# B&R Automation Studio project EFI (part 14)

#### FileManager.st
```iecst
ACTION FileManager:

	CASE Handling.Data.Step OF

		0:  (* link (create) a file device *)
			Handling.Functionblock.DevLink_0.enable := 1;
			Handling.Functionblock.DevLink_0.pDevice := ADR(Handling.Data.Device);  (* name of the device, which is needed for other functionblocks *)
			Handling.Functionblock.DevLink_0.pParam := ADR(Handling.Data.Parameter);  (* devicepath *)
			Handling.Functionblock.DevLink_0;  (* call the function*)

			IF Handling.Functionblock.DevLink_0.status = 0 THEN  (* DevLink successful *)
				Handling.Data.Step := 1;  (* next Step*)
				FolderHandling.Data.Step := 1;  (* next Step*)
			ELSIF Handling.Functionblock.DevLink_0.status = ERR_FUB_BUSY THEN  (* DevLink not finished -> redo *)
				(* Busy *)
			ELSIF Handling.Functionblock.DevLink_0.status = fiERR_SYSTEM THEN  (* DevLink error = fiERR_SYSTEM -> detailed info with function "FileIoGetSysError" *)
				(* get detail errorinformation *)
				Error := FileIoGetSysError();
				(* Goto Error Step *)
				Handling.Data.Step := 255;

				FolderError := FileIoGetSysError();
				FolderHandling.Data.Step := 255;
			ELSE  (* Goto Error Step *)
				Handling.Data.Step := 255;
				FolderHandling.Data.Step := 255;
			END_IF

		1:  (* Wait and comannd step *)
			IF Handling.Command.bCreateFile = 1 THEN
				(* Create a new file with the name from the variable "Handling.Data.FileName" *)
				Handling.Data.Step := 10;  (* next Step*)

			ELSIF Handling.Command.bWriteFile = 1 THEN
				(* writes the data from variable "Handling.Data.WriteData"
				   in the file with the name from the variable "Handling.Data.FileName" *)
				Handling.Data.Step := 20;  (* next Step*)

			ELSIF Handling.Command.bReadFile = 1 THEN
				(* read data to variable "Handling.Data.ReadData"
				   from the file with the name of the variable "Handling.Data.FileName" *)
				Handling.Data.Step := 30;  (* next Step*)

			ELSIF Handling.Command.bReadExFile = 1 THEN
				(* read data to variable "Handling.Data.ReadData"
				   from the file with the name of the variable "Handling.Data.FileName" *)
				Handling.Data.Step := 40;  (* next Step*)

			ELSIF Handling.Command.bCopyFile = 1 THEN
				(* creates a copy with the name from the variable "Handling.Data.NewFileName"
				   from the file with the name from the variable "Handling.Data.FileName" *)
				Handling.Data.Step := 50;  (* next Step*)

			ELSIF Handling.Command.bRenameFile = 1 THEN
				(* renames the the file with the name from the variable "Handling.Data.FileName"
				   to the name from the variable "Handling.Data.NewFileName" *)
				Handling.Data.Step := 60;  (* next Step*)

			ELSIF Handling.Command.bDeleteFile = 1 THEN
				(* deletes the file with the name from the variable "Handling.Data.FileName" *)
				Handling.Data.Step := 70;  (* next Step*)

			END_IF

			(***********************************************************************************************)
		10:  (* create a new File with the selected name  *)
			Handling.Functionblock.FileCreate_0.enable := 1;
			Handling.Functionblock.FileCreate_0.pDevice := ADR(Handling.Data.Device);  (* name of the linked device *)
			Handling.Functionblock.FileCreate_0.pFile := ADR(Handling.Data.FileName);  (* name of the file *)
			Handling.Functionblock.FileCreate_0;  (* call the function*)

			IF Handling.Functionblock.FileCreate_0.status = 0 THEN  (* FileCreate successful *)
				Handling.Data.Step := 11;  (* next Step*)
			ELSIF Handling.Functionblock.FileCreate_0.status = ERR_FUB_BUSY THEN  (* FileCreate not finished -> redo *)
				(* Busy *)
			ELSE  (* Goto Error Step *)
				Handling.Data.Step := 255;
			END_IF

		11:	 (* close file, because of limited number of available file handles on the system *)
			Handling.Functionblock.FileClose_0.enable := 1;
			Handling.Functionblock.FileClose_0.ident := Handling.Functionblock.FileCreate_0.ident; (* ident for FileCreate-functionblock*)
			Handling.Functionblock.FileClose_0;  (* call the function*)

			IF Handling.Functionblock.FileClose_0.status = 0 THEN  (* FileClose successful *)
				Handling.Data.Step := 1;  (* next Step*)
				Handling.Command.bCreateFile := 0;  (* clear command *)
			ELSIF Handling.Functionblock.FileClose_0.status = ERR_FUB_BUSY THEN  (* FileClose not finished -> redo *)
				(* Busy *)
			ELSE  (* Goto Error Step *)
				Handling.Data.Step := 255;
			END_IF

			(***********************************************************************************************)
		20:	(* open file for write access *)
			Handling.Functionblock.FileOpen_0.enable := 1;
			Handling.Functionblock.FileOpen_0.pDevice := ADR(Handling.Data.Device);  (* name of the linked device *)
			Handling.Functionblock.FileOpen_0.pFile :=  ADR(Handling.Data.FileName);  (* name of the file *)
			Handling.Functionblock.FileOpen_0.mode := fiWRITE_ONLY; (* write access *)
			Handling.Functionblock.FileOpen_0;  (* call the function*)

			IF Handling.Functionblock.FileOpen_0.status = 0 THEN  (* FileOpen successful *)
				Handling.Data.Step := 21;  (* next Step*)
			ELSIF Handling.Functionblock.FileOpen_0.status = ERR_FUB_BUSY THEN  (* FileOpen not finished -> redo *)
				(* Busy *)
			ELSE  (* Goto Error Step *)
				Handling.Data.Step := 255;
			END_IF

		21: (* write data into file *)
			Handling.Functionblock.FileWrite_0.enable := 1;
			Handling.Functionblock.FileWrite_0.ident := Handling.Functionblock.FileOpen_0.ident;
			Handling.Functionblock.FileWrite_0.offset := 0; (* start at the beginning of the file *)
			Handling.Functionblock.FileWrite_0.pSrc := ADR(Handling.Data.WriteData);
			Handling.Functionblock.FileWrite_0.len := strlen( ADR(Handling.Data.WriteData) );
			Handling.Functionblock.FileWrite_0;  (* call the function*)

			IF Handling.Functionblock.FileWrite_0.status = 0 THEN  (* FileWrite successful *)
				Handling.Data.Step := 22;  (* next Step*)
			ELSIF Handling.Functionblock.FileWrite_0.status = ERR_FUB_BUSY THEN  (* FileWrite not finished -> redo *)
				(* Busy *)
			ELSE  (* Goto Error Step *)
				Handling.Data.Step := 255;
			END_IF

		22:	 (* close file, because of limited number of available file handles on the system *)
			Handling.Functionblock.FileClose_0.enable := 1;
			Handling.Functionblock.FileClose_0.ident := Handling.Functionblock.FileOpen_0.ident; (* ident for FileCreate-functionblock*)
			Handling.Functionblock.FileClose_0;  (* call the function*)

			IF Handling.Functionblock.FileClose_0.status = 0 THEN  (* FileClose successful *)
				Handling.Data.Step := 1;  (* next Step*)
				Handling.Command.bWriteFile := 0;  (* clear command *)
			ELSIF Handling.Functionblock.FileClose_0.status = ERR_FUB_BUSY THEN  (* FileClose not finished -> redo *)
				(* Busy *)
			ELSE  (* Goto Error Step *)
				Handling.Data.Step := 255;
			END_IF

			(***********************************************************************************************)
		30:	(* open file for read access *)
			Handling.Functionblock.FileOpen_0.enable := 1;
			Handling.Functionblock.FileOpen_0.pDevice := ADR(Handling.Data.Device);  (* name of the linked device *)
			Handling.Functionblock.FileOpen_0.pFile :=  ADR(Handling.Data.FileName);  (* name of the file *)
			Handling.Functionblock.FileOpen_0.mode := fiREAD_ONLY;  (* read access *)
			Handling.Functionblock.FileOpen_0;  (* call the function*)

			IF Handling.Functionblock.FileOpen_0.status = 0 THEN  (* FileOpen successful *)
				Handling.Data.Step := 31;  (* next Step*)
			ELSIF Handling.Functionblock.FileOpen_0.status = ERR_FUB_BUSY THEN  (* FileOpen not finished -> redo *)
				(* Busy *)
			ELSE  (* Goto Error Step *)
				Handling.Data.Step := 255;
			END_IF

		31: (* read data from file *)
			Handling.Functionblock.FileRead_0.enable := 1;
			Handling.Functionblock.FileRead_0.ident := Handling.Functionblock.FileOpen_0.ident;  (* ident of the previous "FileOpen" *)
			Handling.Functionblock.FileRead_0.offset := 0;  (* start at the beginning of the file *)
			Handling.Functionblock.FileRead_0.pDest := ADR(Handling.Data.ReadData);  (* adress of the destination of reaaded datas *)
			Handling.Functionblock.FileRead_0.len := SIZEOF( Handling.Data.ReadData );  (* lenght of data, which should be readed *)
			Handling.Functionblock.FileRead_0;  (* call the function*)

			IF Handling.Functionblock.FileRead_0.status = 0 THEN  (* FileRead successful *)
				Handling.Data.Step := 32;  (* next Step*)
			ELSIF Handling.Functionblock.FileRead_0.status = ERR_FUB_BUSY THEN  (* FileRead not finished -> redo *)
				(* Busy *)
			ELSE  (* Goto Error Step *)
				Handling.Data.Step := 255;
			END_IF

		32:	 (* close file, because of limited number of available file handles on the system *)
			Handling.Functionblock.FileClose_0.enable := 1;
			Handling.Functionblock.FileClose_0.ident := Handling.Functionblock.FileOpen_0.ident; (* ident for FileCreate-functionblock*)
			Handling.Functionblock.FileClose_0;  (* call the function*)

			IF Handling.Functionblock.FileClose_0.status = 0 THEN  (* FileClose successful *)
				Handling.Data.Step := 1;  (* next Step*)
				Handling.Command.bReadFile := 0;  (* clear command *)
			ELSIF Handling.Functionblock.FileClose_0.status = ERR_FUB_BUSY THEN  (* FileClose not finished -> redo *)
				(* Busy *)
			ELSE  (* Goto Error Step *)
				Handling.Data.Step := 255;
			END_IF

			(***********************************************************************************************)
		40:	(* open file for read access *)
			Handling.Functionblock.FileOpen_0.enable := 1;
			Handling.Functionblock.FileOpen_0.pDevice := ADR(Handling.Data.Device);  (* name of the linked device *)
			Handling.Functionblock.FileOpen_0.pFile :=  ADR(Handling.Data.FileName);  (* name of the file *)
			Handling.Functionblock.FileOpen_0.mode := fiREAD_ONLY;  (* read access *)
			Handling.Functionblock.FileOpen_0;  (* call the function*)

			IF Handling.Functionblock.FileOpen_0.status = 0 THEN  (* FileOpen successful *)
				Handling.Data.Step := 41;  (* next Step*)
			ELSIF Handling.Functionblock.FileOpen_0.status = ERR_FUB_BUSY THEN  (* FileOpen not finished -> redo *)
				(* Busy *)
			ELSE  (* Goto Error Step *)
				Handling.Data.Step := 255;
			END_IF

		41: (* read data from file *)
			Handling.Functionblock.FileReadEx_0.enable := 1;
			Handling.Functionblock.FileReadEx_0.ident := Handling.Functionblock.FileOpen_0.ident;  (* ident of the previous "FileOpen" *)
			Handling.Functionblock.FileReadEx_0.offset := 0;  (* start at the beginning of the file *)
			Handling.Functionblock.FileReadEx_0.pDest := ADR(Handling.Data.ReadData);  (* adress of the destination of reaaded datas *)
			Handling.Functionblock.FileReadEx_0.len := SIZEOF( Handling.Data.ReadData );  (* lenght of data, which should be readed *)
			Handling.Functionblock.FileReadEx_0;  (* call the function*)

			IF Handling.Functionblock.FileReadEx_0.status = 0 THEN  (* FileReadEx successful *)
				(* Handling.Functionblock.FileReadEx_0.bytesread includes the lenght of the readed data *)
				Handling.Data.Step := 42;  (* next Step*)
			ELSIF Handling.Functionblock.FileReadEx_0.status = ERR_FUB_BUSY THEN  (* FileReadEx not finished -> redo *)
				(* Busy *)
			ELSE  (* Goto Error Step *)
				Handling.Data.Step := 255;
			END_IF

		42:	 (* close file, because of limited number of available file handles on the system *)
			Handling.Functionblock.FileClose_0.enable := 1;
			Handling.Functionblock.FileClose_0.ident := Handling.Functionblock.FileOpen_0.ident; (* ident for FileCreate-functionblock*)
			Handling.Functionblock.FileClose_0;  (* call the function*)

			IF Handling.Functionblock.FileClose_0.status = 0 THEN  (* FileClose successful *)
				Handling.Data.Step := 1;  (* next Step*)
				Handling.Command.bReadExFile := 0;  (* clear command *)
			ELSIF Handling.Functionblock.FileClose_0.status = ERR_FUB_BUSY THEN  (* FileClose not finished -> redo *)
				(* Busy *)
			ELSE  (* Goto Error Step *)
				Handling.Data.Step := 255;
			END_IF

			(***********************************************************************************************)
		50: (* copy a file *)

			Handling.Functionblock.FileCopy_0.enable := 1;
			Handling.Functionblock.FileCopy_0.option := fiOVERWRITE;  (* overwrite existing file *)
			Handling.Functionblock.FileCopy_0.pSrcDev := ADR(Handling.Data.Device);  (* name of a linked device *)
			Handling.Functionblock.FileCopy_0.pSrc := ADR(Handling.Data.FileName);  (* name of the source file *)
			Handling.Functionblock.FileCopy_0.pDestDev := ADR(Handling.Data.Device);  (* name of a linked device *)
			Handling.Functionblock.FileCopy_0.pDest := ADR(Handling.Data.NewFileName);  (* name of the new file*)
			Handling.Functionblock.FileCopy_0;  (* call the function*)

			IF Handling.Functionblock.FileCopy_0.status = 0 THEN  (* FileCopy successful *)
				Handling.Data.Step := 1;  (* next Step*)
				Handling.Command.bCopyFile := 0;  (* clear command *)
			ELSIF Handling.Functionblock.FileCopy_0.status = ERR_FUB_BUSY THEN  (* FileCopy not finished -> redo *)
				(* Busy *)
			ELSE  (* Goto Error Step *)
				Handling.Data.Step := 255;
			END_IF

			(***********************************************************************************************)
		60: (* rename a file *)

			Handling.Functionblock.FileRename_0.enable := 1;
			Handling.Functionblock.FileRename_0.pDevice := ADR(Handling.Data.Device);  (* name of the linked device *)
			Handling.Functionblock.FileRename_0.pName := ADR(Handling.Data.FileName);  (* actual file name *)
			Handling.Functionblock.FileRename_0.pNewName := ADR(Handling.Data.NewFileName);  (* new file name *)
			Handling.Functionblock.FileRename_0;  (* call the function*)

			IF Handling.Functionblock.FileRename_0.status = 0 THEN  (* FileRename successful *)
				Handling.Data.Step := 1;  (* next Step*)
				Handling.Command.bRenameFile := 0;  (* clear command *)
			ELSIF Handling.Functionblock.FileRename_0.status = ERR_FUB_BUSY THEN  (* FileRename not finished -> redo *)
				(* Busy *)
			ELSE  (* Goto Error Step *)
				Handling.Data.Step := 255;
			END_IF

			(***********************************************************************************************)
		70: (* delete a file *)

			Handling.Functionblock.FileDelete_0.enable := 1;
			Handling.Functionblock.FileDelete_0.pDevice := ADR(Handling.Data.Device);  (* name of a linked device *)
			Handling.Functionblock.FileDelete_0.pName := ADR(Handling.Data.FileName);  (* name of the source file *)
			Handling.Functionblock.FileDelete_0;  (* call the function*)

			IF Handling.Functionblock.FileDelete_0.status = 0 THEN  (* FileRename successful *)
				Handling.Data.Step := 1;  (* next Step*)
				Handling.Command.bDeleteFile := 0;  (* clear command *)
			ELSIF Handling.Functionblock.FileDelete_0.status = ERR_FUB_BUSY THEN  (* FileRename not finished -> redo *)
				(* Busy *)
			ELSE  (* Goto Error Step *)
				Handling.Data.Step := 255;
			END_IF

			(***********************************************************************************************)
		255:  (* Here some error Handling has to be implemented *)

	END_CASE

END_ACTION
```

#### FolderManager.st
```iecst
ACTION FolderManager:

	CASE FolderHandling.Data.Step OF

		0:  (* link (create) a file device *)
			//			FolderHandling.Functionblock.DevLink_0.enable := 1;
			//			FolderHandling.Functionblock.DevLink_0.pDevice := ADR(FolderHandling.Data.Device);  (* name of the device, which is needed for other functionblocks *)
			//			FolderHandling.Functionblock.DevLink_0.pParam := ADR(FolderHandling.Data.Parameter);  (* devicepath *)
			//			FolderHandling.Functionblock.DevLink_0;  (* call the function*)
			//
			//			IF FolderHandling.Functionblock.DevLink_0.status = 0 THEN  (* DevLink successful *)
			//				FolderHandling.Data.Step := 1;  (* next Step*)
			//			ELSIF FolderHandling.Functionblock.DevLink_0.status = ERR_FUB_BUSY THEN  (* DevLink not finished -> redo *)
			//				(* Busy *)
			//			ELSIF FolderHandling.Functionblock.DevLink_0.status = fiERR_SYSTEM THEN  (* DevLink FolderError = fiERR_SYSTEM -> detailed info with function "FileIoGetSysFolderError" *)
			//				(* get detail FolderErrorinformation *)
			//				FolderError := FileIoGetSysFolderError();
			//				(* Goto FolderError Step *)
			//				FolderHandling.Data.Step := 255;
			//			ELSE  (* Goto FolderError Step *)
			//				FolderHandling.Data.Step := 255;
			//			END_IF

		1:  (* Wait and comannd step *)
			IF FolderHandling.Command.bDirRead = 1 THEN
				(* read all names of files and folders into the string-array "FolderHandling.Data.FileList" *)
				FolderHandling.Data.Step := 10;  (* next Step*)

			ELSIF FolderHandling.Command.bDirCreate = 1 THEN
				(* creates a new directory with the name on the variable "FolderHandling.Data.DirName" *)
				FolderHandling.Data.Step := 20;  (* next Step*)

			ELSIF FolderHandling.Command.bDirCopy = 1 THEN
				(* copy a directory with the name on the variable "FolderHandling.Data.DirName"
				   to a directory with the name on the variable "FolderHandling.Data.NewDirName"*)
				FolderHandling.Data.Step := 30;  (* next Step*)

			ELSIF FolderHandling.Command.bDirRename = 1 THEN
				(* rename the directory with the name on the variable "FolderHandling.Data.DirName"
				   to the name on the variable "FolderHandling.Data.NewDirName"*)
				FolderHandling.Data.Step := 40;  (* next Step*)

			ELSIF FolderHandling.Command.bDirDelete = 1 THEN
				(* delete the directory with the name on the variable "FolderHandling.Data.DirName" *)
				FolderHandling.Data.Step := 50;  (* next Step*)

			ELSIF FolderHandling.Command.bDevMemInfo = 1 THEN
				(* read information about your device *)
				FolderHandling.Data.Step := 60;  (* next Step*)

			ELSIF FolderHandling.Command.bGetAttributes = 1 THEN
				(* read information about your device-settings *)
				FolderHandling.Data.Step := 70;  (* next Step*)

			ELSIF FolderHandling.Command.bSetAttributes = 1 THEN
				(* set device settings*)
				FolderHandling.Data.Step := 80;  (* next Step*)

			END_IF

			(***********************************************************************************************)
		10: (* calulate the number of files and directories *)
			FolderHandling.Functionblock.DirInfo_0.enable := 1;
			FolderHandling.Functionblock.DirInfo_0.pDevice := ADR(FolderHandling.Data.Device);  (* name of the device *)
			FolderHandling.Functionblock.DirInfo_0.pPath := 0;
			FolderHandling.Functionblock.DirInfo_0;  (* call the function*)

			IF FolderHandling.Functionblock.DirInfo_0.status = 0 THEN  (* DirInfo successful *)
				(* FolderHandling.Functionblock.DirInfo_0.dirnum contains the number of found folders *)
				(* FolderHandling.Functionblock.DirInfo_0.filenum contains the number of found files *)
				FolderCounter := 0;  (* reset FolderCounter *)
				memset( ADR(FolderHandling.Data.FileList[0]), 0, SIZEOF(FolderHandling.Data.FileList) );  (* clear list*)
				FolderHandling.Data.Step := 11;  (* next step*)
			ELSIF FolderHandling.Functionblock.DirInfo_0.status = ERR_FUB_BUSY THEN  (* DirInfo not finished -> redo *)
				(* Busy *)
			ELSE  (* Goto FolderError Step *)
				FolderHandling.Data.Step := 255;
			END_IF

			(***********************************************************************************************)
		11: (* read information about files and folders *)
			FolderHandling.Functionblock.DirRead_0.enable := 1;
			FolderHandling.Functionblock.DirRead_0.pDevice := ADR(FolderHandling.Data.Device);  (* name of the device *)
			FolderHandling.Functionblock.DirRead_0.pPath := 0;
			FolderHandling.Functionblock.DirRead_0.option := fiBOTH;  (* read files and folders *)
			FolderHandling.Functionblock.DirRead_0.entry := FolderCounter;
			FolderHandling.Functionblock.DirRead_0.pData := ADR(ReadData);
			FolderHandling.Functionblock.DirRead_0.data_len := SIZEOF(ReadData);
			FolderHandling.Functionblock.DirRead_0;  (* call the function*)

			IF FolderHandling.Functionblock.DirRead_0.status = 0 THEN  (* DirRead successful *)
				(* copy found name into string-array *)
				strcpy( ADR(FolderHandling.Data.FileList[FolderCounter]), ADR(ReadData.Filename[0]) );
				(* increase FolderCounter *)
				FolderCounter := FolderCounter + 1;
				(* are all files and folders readed out? *)
				IF ( FolderCounter < (FolderHandling.Functionblock.DirInfo_0.dirnum + FolderHandling.Functionblock.DirInfo_0.filenum) ) THEN
					FolderHandling.Data.Step := 11;  (* read next element *)
				ELSE
					FolderHandling.Data.Step := 1;  (* next step *)
					FolderHandling.Command.bDirRead := 0; (* reset command *)
				END_IF
			ELSIF FolderHandling.Functionblock.DirRead_0.status = ERR_FUB_BUSY THEN  (* DirRead not finished -> redo *)
				(* Busy *)
			ELSE  (* Goto FolderError Step *)
				FolderHandling.Data.Step := 255;
			END_IF

			(***********************************************************************************************)
		20: (* create a new folder *)
			FolderHandling.Functionblock.DirCreate_0.enable := 1;
			FolderHandling.Functionblock.DirCreate_0.pDevice := ADR(FolderHandling.Data.Device);  (* name of the device *)
			FolderHandling.Functionblock.DirCreate_0.pName := ADR(FolderHandling.Data.DirName);
			FolderHandling.Functionblock.DirCreate_0;  (* call the function*)

			IF FolderHandling.Functionblock.DirCreate_0.status = 0 THEN  (* DirCreate successful *)
				FolderHandling.Data.Step := 1;  (* next step *)
				FolderHandling.Command.bDirCreate := 0; (* reset command *)
			ELSIF FolderHandling.Functionblock.DirCreate_0.status = ERR_FUB_BUSY THEN  (* DirCreate not finished -> redo *)
				(* Busy *)
			ELSE  (* Goto FolderError Step *)
				FolderHandling.Data.Step := 255;
			END_IF

			(***********************************************************************************************)
		30: (* copy a folder *)
			FolderHandling.Functionblock.DirCopy_0.enable := 1;
			FolderHandling.Functionblock.DirCopy_0.pSrcDev := ADR(FolderHandling.Data.Device);  (* name of the device *)
			FolderHandling.Functionblock.DirCopy_0.pSrcDir := ADR(FolderHandling.Data.DirName);  (* source folder name *)
			FolderHandling.Functionblock.DirCopy_0.pDestDev := ADR(FolderHandling.Data.Device);  (* name of the device *)
			FolderHandling.Functionblock.DirCopy_0.pDestDir := ADR(FolderHandling.Data.NewDirName);  (* destination folder name *)
			FolderHandling.Functionblock.DirCopy_0.option := fiOVERWRITE; (* overwrite mode*)
			FolderHandling.Functionblock.DirCopy_0;  (* call the function*)

			IF FolderHandling.Functionblock.DirCopy_0.status = 0 THEN  (* DirCopy successful *)
				FolderHandling.Data.Step := 1;  (* next step *)
				FolderHandling.Command.bDirCopy := 0; (* reset command *)
			ELSIF FolderHandling.Functionblock.DirCopy_0.status = ERR_FUB_BUSY THEN  (* DirCopy not finished -> redo *)
				(* Busy *)
			ELSE  (* Goto FolderError Step *)
				FolderHandling.Data.Step := 255;
			END_IF

			(***********************************************************************************************)
		40: (* rename a folder *)
			FolderHandling.Functionblock.DirRename_0.enable := 1;
			FolderHandling.Functionblock.DirRename_0.pDevice := ADR(FolderHandling.Data.Device);  (* name of the device *)
			FolderHandling.Functionblock.DirRename_0.pName:= ADR(FolderHandling.Data.DirName);  (* name of the folder *)
			FolderHandling.Functionblock.DirRename_0.pNewName := ADR(FolderHandling.Data.NewDirName);  (* new name of the folder*)
			FolderHandling.Functionblock.DirRename_0;  (* call the function*)

			IF FolderHandling.Functionblock.DirRename_0.status = 0 THEN  (* DirRename successful *)
				FolderHandling.Data.Step := 1;  (* next step *)
				FolderHandling.Command.bDirRename := 0; (* reset command *)
			ELSIF FolderHandling.Functionblock.DirRename_0.status = ERR_FUB_BUSY THEN  (* DirRename not finished -> redo *)
				(* Busy *)
			ELSE  (* Goto FolderError Step *)
				FolderHandling.Data.Step := 255;
			END_IF

			(***********************************************************************************************)
		50: (* delete a folder *)
			FolderHandling.Functionblock.DirDelete_0.enable := 1;
			FolderHandling.Functionblock.DirDelete_0.pDevice := ADR(FolderHandling.Data.Device);  (* name of the device *)
			FolderHandling.Functionblock.DirDelete_0.pName:= ADR(FolderHandling.Data.DirName);  (* name of the folder *)
			FolderHandling.Functionblock.DirDelete_0;  (* call the function*)

			IF FolderHandling.Functionblock.DirDelete_0.status = 0 THEN  (* DirDelete successful *)
				FolderHandling.Data.Step := 1;  (* next step *)
				FolderHandling.Command.bDirDelete := 0; (* reset command *)
			ELSIF FolderHandling.Functionblock.DirDelete_0.status = ERR_FUB_BUSY THEN  (* DirDelete not finished -> redo *)
				(* Busy *)
			ELSE  (* Goto FolderError Step *)
				FolderHandling.Data.Step := 255;
			END_IF

			(***********************************************************************************************)
		60: (* read information about your device *)
			FolderHandling.Functionblock.DevMemInfo_0.enable := 1;
			FolderHandling.Functionblock.DevMemInfo_0.pDevice := ADR(FolderHandling.Data.Device);  (* name of the device *)
			FolderHandling.Functionblock.DevMemInfo_0;  (* call the function*)

			IF FolderHandling.Functionblock.DevMemInfo_0.status = 0 THEN  (* DevMemInfo successful *)
				(* FolderHandling.Functionblock.DevMemInfo_0.memsize contains the memsize of your device *)
				(* FolderHandling.Functionblock.DevMemInfo_0.freemem contains the free memsize of your device*)
				FolderHandling.Data.Step := 1;  (* next step *)
				FolderHandling.Command.bDevMemInfo := 0; (* reset command *)
			ELSIF FolderHandling.Functionblock.DevMemInfo_0.status = ERR_FUB_BUSY THEN  (* DevMemInfo not finished -> redo *)
				(* Busy *)
			ELSE  (* Goto FolderError Step *)
				FolderHandling.Data.Step := 255;
			END_IF

			(***********************************************************************************************)
		70: (* read information about your device settings *)
			FolderHandling.Functionblock.GetAttributes_0.enable := 1;
			FolderHandling.Functionblock.GetAttributes_0.pDevice := ADR(FolderHandling.Data.Device);  (* name of the device *)
			FolderHandling.Functionblock.GetAttributes_0.pPath := ADR(FolderHandling.Data.DirName);  (* name of the folder *)
			FolderHandling.Functionblock.GetAttributes_0;  (* call the function*)

			IF FolderHandling.Functionblock.GetAttributes_0.status = 0 THEN  (* GetAttributes successful *)
				(* FolderHandling.Functionblock.GetAttributes_0.attributes *)
				FolderHandling.Data.Step := 1;  (* next step *)
				FolderHandling.Command.bGetAttributes := 0; (* reset command *)
			ELSIF FolderHandling.Functionblock.GetAttributes_0.status = ERR_FUB_BUSY THEN  (* GetAttributes not finished -> redo *)
				(* Busy *)
			ELSE  (* Goto FolderError Step *)
				FolderHandling.Data.Step := 255;
			END_IF

			(***********************************************************************************************)
		80: (* set device settings *)
			FolderHandling.Functionblock.SetAttributes_0.enable := 1;
			FolderHandling.Functionblock.SetAttributes_0.pDevice := ADR(FolderHandling.Data.Device);  (* name of the device *)
			FolderHandling.Functionblock.SetAttributes_0.pPath := ADR(FolderHandling.Data.DirName);  (* name of the folder *)
			FolderHandling.Functionblock.SetAttributes_0.attributes := fiATTR_RDONLY;  (* make device readonly *)
			FolderHandling.Functionblock.SetAttributes_0.option := fiRECURSIVE;  (* include all subfolders *)
			FolderHandling.Functionblock.SetAttributes_0;  (* call the function*)

			IF FolderHandling.Functionblock.SetAttributes_0.status = 0 THEN  (* GetAttributes successful *)
				(* FolderHandling.Functionblock.GetAttributes_0.attributes *)
				FolderHandling.Data.Step := 1;  (* next step *)
				FolderHandling.Command.bSetAttributes := 0; (* reset command *)
			ELSIF FolderHandling.Functionblock.SetAttributes_0.status = ERR_FUB_BUSY THEN  (* GetAttributes not finished -> redo *)
				(* Busy *)
			ELSE  (* Goto FolderError Step *)
				FolderHandling.Data.Step := 255;
			END_IF

			(***********************************************************************************************)
		255:  (* Here some FolderError FolderHandling has to be implemented *)

	END_CASE

END_ACTION
```

#### RegFileName.st
```iecst
ACTION GetSystemTime:

	getTime.enable := TRUE;
	getTime.pDTStructure := ADR(TimeValue);
	getTime();

	IF getTime.status = ERR_OK THEN
		iYear := TimeValue.year;
		brsitoa(iYear, ADR(strYear));
	END_IF

END_ACTION

ACTION CreateFolderYear:

	strcpy( ADR(FolderHandling.Data.DirName), ADR(FOLDER_SIM_REG) );
	brsstrcat( ADR(FolderHandling.Data.DirName), ADR('/'));
	brsstrcat( ADR(FolderHandling.Data.DirName), ADR(strYear));

END_ACTION

ACTION CreateFileReg:

	strcpy( ADR(Handling.Data.FileName), ADR(FOLDER_SIM_REG) );
	brsstrcat( ADR(Handling.Data.FileName), ADR('/'));
	brsstrcat( ADR(Handling.Data.FileName), ADR(strYear));
	brsstrcat( ADR(Handling.Data.FileName), ADR('/'));

	brsitoa(iYear, ADR(FileNameAux));
	brsstrcat( ADR(Handling.Data.FileName), ADR(FileNameAux));
	brsstrcat( ADR(Handling.Data.FileName), ADR('-'));

	FileNameAuxPre := '0';
	iDigits := brsitoa(TimeValue.month, ADR(FileNameAux));
	IF iDigits = 1 THEN
		brsstrcat( ADR(FileNameAuxPre), ADR(FileNameAux));
		brsstrcat( ADR(Handling.Data.FileName), ADR(FileNameAuxPre));
	ELSE
		brsstrcat( ADR(Handling.Data.FileName), ADR(FileNameAux));
	END_IF
	brsstrcat( ADR(Handling.Data.FileName), ADR('-'));

	FileNameAuxPre := '0';
	iDigits := brsitoa(TimeValue.day, ADR(FileNameAux));
	IF iDigits = 1 THEN
		brsstrcat( ADR(FileNameAuxPre), ADR(FileNameAux));
		brsstrcat( ADR(Handling.Data.FileName), ADR(FileNameAuxPre));
	ELSE
		brsstrcat( ADR(Handling.Data.FileName), ADR(FileNameAux));
	END_IF
	brsstrcat( ADR(Handling.Data.FileName), ADR('.'));

	FileNameAuxPre := '0';
	iDigits := brsitoa(TimeValue.hour, ADR(FileNameAux));
	IF iDigits = 1 THEN
		brsstrcat( ADR(FileNameAuxPre), ADR(FileNameAux));
		brsstrcat( ADR(Handling.Data.FileName), ADR(FileNameAuxPre));
	ELSE
		brsstrcat( ADR(Handling.Data.FileName), ADR(FileNameAux));
	END_IF
	brsstrcat( ADR(Handling.Data.FileName), ADR('-'));

	brsstrcat( ADR(Handling.Data.FileName), ADR('00')); //For the minutes

END_ACTION
```

#### SimUseRegister.st
```iecst
(********************************************************************
 * COPYRIGHT -- EFI
 ********************************************************************
 * Program: SimUseRegister
 * File: SimUseRegister.st
 * Author: Jorge Murria
 * Created: February 03, 2022
 ********************************************************************
 * Implementation of program SimUseRegister
 ********************************************************************)

(******************************************)
(* init program                           *)
(******************************************)
PROGRAM _INIT

	(* device name for different function blocks needed (choose yourself) *)
	strcpy( ADR(Handling.Data.Device), ADR('LOCAL_DEVICE') );
	(* perameter string, layout see in the online help by function block "devlink" *)
	strcpy( ADR(Handling.Data.Parameter), ADR('"/DEVICE=C:/BrAutomation') );

	//Connect Both Handlers
	FolderHandling.Data.Device := Handling.Data.Device;
	FolderHandling.Data.Parameter := Handling.Data.Parameter;

END_PROGRAM

(******************************************)
(* cyclic program                         *)
(******************************************)
PROGRAM _CYCLIC

	GetSystemTime;

	//To avoid start the process with wrong data
	IF iYear = 0 THEN
		RETURN;
	END_IF

	CASE SimRegState OF
		SIMR_STOPPED:
			SimRegState := SIMR_IDLE;

		SIMR_IDLE:
			SimRegState := SIMR_CREATE_MAIN;

		SIMR_CREATE_MAIN:
			strcpy( ADR(FolderHandling.Data.DirName), ADR(FOLDER_SIM_REG) );

			FolderHandling.Command.bDirCreate := TRUE;
			SimRegState := SIMR_CREATING_MAIN;

		SIMR_CREATING_MAIN:
			xFunctionEnded := FolderHandling.Functionblock.DirCreate_0.status = ERR_OK OR FolderHandling.Functionblock.DirCreate_0.status = fiERR_DIR_ALREADY_EXIST;
			xStepManaged := FolderHandling.Data.Step = 1 OR FolderHandling.Data.Step = 255;
			IF  xFunctionEnded AND xStepManaged THEN
				FolderHandling.Data.Step := 1; //If the folder exists, remove the error
				SimRegState := SIMR_CREATE_YEAR;
			END_IF

		SIMR_CREATE_YEAR:
			CreateFolderYear;

			FolderHandling.Command.bDirCreate := TRUE;
			SimRegState := SIMR_CREATING_YEAR;

		SIMR_CREATING_YEAR:
			xFunctionEnded := FolderHandling.Functionblock.DirCreate_0.status = ERR_OK OR FolderHandling.Functionblock.DirCreate_0.status = fiERR_DIR_ALREADY_EXIST;
			xStepManaged := FolderHandling.Data.Step = 1 OR FolderHandling.Data.Step = 255;
			IF  xFunctionEnded AND xStepManaged THEN
				FolderHandling.Data.Step := 1; //If the folder exists, remove the error
				SimRegState := SIMR_CREATE_FILEREG;
			END_IF

		SIMR_CREATE_FILEREG:
			CreateFileReg;
			lastHour := TimeValue.hour;

			Handling.Command.bCreateFile := TRUE;
			SimRegState := SIMR_CREATING_FILEREG;

		SIMR_CREATING_FILEREG:
			xFunctionEnded := Handling.Functionblock.FileCreate_0.status = ERR_OK OR Handling.Functionblock.FileCreate_0.status = fiERR_EXIST;
			xStepManaged := Handling.Data.Step = 1 OR Handling.Data.Step = 255;
			IF  xFunctionEnded AND xStepManaged THEN
				Handling.Data.Step := 1; //If the folder exists, remove the error
				SimRegState := SIMR_IDLE_MAIN;
			END_IF

		SIMR_IDLE_MAIN:
			//Every new our, Register and write a new file
			IF lastHour <> TimeValue.hour THEN
				SimRegState := SIMR_CREATE_YEAR;
			END_IF

	END_CASE;

	FileManager;

	FolderManager;

END_PROGRAM
```

### Program Logical/ExtPack/_Tools/TestBench/TraySim/TraySim_v1/TraySim (IEC)

#### TraySim.var - Local variables
```iecst
VAR
	trayData : REFERENCE TO stTraySim;
	ton_ToOut : TON;
	ton_ToIn : TON;
	ton_ReboundOut : TON;
	ton_ReboundIn : TON;
	xReboundedOut : BOOL;
	xReboundedIn : BOOL;
END_VAR
```

### TraySim.typ - Local data types
```iecst
TYPE
	stTrayCmd : 	STRUCT
		ToOut : BOOL;
		ToIn : BOOL;
		ReboundToOut : BOOL; (*The signal appears at the end but desappears just after appear*)
		ReboundToIn : BOOL; (*The signal appears at the end but desappears just after appear*)
		UnplugInSensor : BOOL; (*Command to unplug IN sensor*)
		UnplugOutSensor : BOOL; (*Command to unplug OUT sensor*)
		ResetOut : BOOL; (*EDGE Command to reset the signal. Reseted in the element*)
		ResetIn : BOOL; (*EDGE Command to reset the signal. Reseted in the element*)
	END_STRUCT;
	stTrayState : 	STRUCT
		OutPosition : BOOL;
		InPosition : BOOL;
	END_STRUCT;
	stTraySim : 	STRUCT
		State : stTrayState;
		Commands : stTrayCmd;
	END_STRUCT;
END_TYPE
```

- BeltCleaning.graphml (not shown)

### Program Logical/ExtPack/_Transport/BeltCleaning/BeltCleaning_v1/BeltCleaning (IEC)

#### BeltCleaning.st - Init, cyclic, exit code
```iecst
PROGRAM _INIT
	(* Insert code here *)

END_PROGRAM

PROGRAM _CYCLIC

	//NOZOMITWO-1912

	dataBeltClean ACCESS ADR (gBeltClean);

	IF NOT dataBeltClean.Parameters.xInstalled THEN
		dataBeltClean.Outputs := ResetOutputs;
		dataBeltClean.Status.State := BCLEAN_NOT_INSTALLED;
		dataBeltClean.Alarm := ResetAlarms;
		dataBeltClean.AlSummary := ResetAlSummary;
		RETURN;
	END_IF

	Alarms;
	AlarmsSummary;
	GeneralLogic;

	CASE dataBeltClean.Status.State OF
		BCLEAN_NOT_INSTALLED:
			IF dataBeltClean.Parameters.xInstalled THEN
				dataBeltClean.Status.State := BCLEAN_DISABLED;
			END_IF

		BCLEAN_FAULT:
			IF NOT dataBeltClean.AlSummary.xAnyAlarm THEN
				dataBeltClean.Status.State := BCLEAN_DISABLED;
			END_IF

		BCLEAN_DISABLED:
			IF dataBeltClean.ParSw.xEnabledByPieces OR dataBeltClean.ParSw.xEnabledByTime THEN
				dataBeltClean.Status.State := BCLEAN_ENABLED;
			ELSIF dataBeltClean.Status.xCleanForced THEN
				dataBeltClean.Status.State := BCLEAN_WAITING_TO_CLEAN;
			END_IF

		BCLEAN_ENABLED:
			IF dataBeltClean.Status.xCleanReqByTime OR dataBeltClean.Status.xCleanReqByPieces THEN
				dataBeltClean.Status.State := BCLEAN_WAITING_SW_CONF;
			ELSIF dataBeltClean.Status.xCleanForced THEN
				dataBeltClean.Status.State := BCLEAN_WAITING_TO_CLEAN;
			ELSIF NOT dataBeltClean.ParSw.xEnabledByPieces AND NOT dataBeltClean.ParSw.xEnabledByTime THEN
				dataBeltClean.Status.State := BCLEAN_DISABLED;
			END_IF

		BCLEAN_WAITING_SW_CONF:
			IF dataBeltClean.CommandsSw.xAcceptRequest OR ton_SwCleanRequest.Q THEN
				dataBeltClean.Status.State := BCLEAN_WAITING_TO_CLEAN;
			ELSIF dataBeltClean.CommandsSw.xRefuseRequest THEN
				ResetCountersAndTimers;
				dataBeltClean.Status.State := BCLEAN_DISABLED;
			END_IF

		BCLEAN_WAITING_TO_CLEAN:
			IF dataBeltClean.Commands.xAcceptRequest AND dataBeltClean.Parameters.xBeltEmpty THEN
				ResetCountersAndTimers;
				dataBeltClean.Status.State := BCLEAN_CLEANING;
			END_IF

		BCLEAN_CLEANING:
			IF ton_Cleaning.Q THEN
				dataBeltClean.Status.State := BCLEAN_DRYING;
			END_IF

		BCLEAN_DRYING:
			IF ton_Drying.Q THEN
				dataBeltClean.Status.State := BCLEAN_DISABLED;
			END_IF

	END_CASE

	dataBeltClean.Status.xCleanRequested := dataBeltClean.Status.State = BCLEAN_WAITING_TO_CLEAN;
	dataBeltClean.Status.xCleanRequestedSw := dataBeltClean.Status.State = BCLEAN_WAITING_SW_CONF;
	dataBeltClean.Status.xCleaning := dataBeltClean.Status.State = BCLEAN_CLEANING OR dataBeltClean.Status.State = BCLEAN_DRYING;

	IF dataBeltClean.Parameters.Mode.xZero THEN
		dataBeltClean.Status.State := BCLEAN_DISABLED;
	ELSIF dataBeltClean.AlSummary.xAlarmStop THEN
		dataBeltClean.Status.State := BCLEAN_FAULT;
	END_IF

	Outputs;

	dataBeltClean.Commands := ResetCommands;
	dataBeltClean.CommandsSw := ResetCommandsSw;

END_PROGRAM
```

#### AlarmsSummary.st
```iecst
ACTION AlarmsSummary:

	dataBeltClean.AlSummary.iReasonWarning.0 := dataBeltClean.Alarm.xAirTurbDisabled;
	dataBeltClean.AlSummary.iReasonWarning.1 := dataBeltClean.Alarm.xAirTurbDisVSDFault;
	dataBeltClean.AlSummary.iReasonWarning.2 := dataBeltClean.Alarm.xBeltNotEmptyToClean;

	dataBeltClean.AlSummary.xAnyWarning := dataBeltClean.AlSummary.iReasonWarning > 0;

	dataBeltClean.AlSummary.iReasonStop[0].0 := dataBeltClean.Alarm.xBeltIsNotRuning;
	dataBeltClean.AlSummary.iReasonStop[0].1 := dataBeltClean.Alarm.xAirTurbEnVSDFault;
	dataBeltClean.AlSummary.iReasonStop[0].2 := dataBeltClean.Alarm.xWaitingToCleanState;
	dataBeltClean.AlSummary.iReasonStop[0].3 := dataBeltClean.Alarm.xBeltIsNotEmpty;

	dataBeltClean.AlSummary.xAlarmStop := dataBeltClean.AlSummary.iReasonStop[0] > 0;

	dataBeltClean.AlSummary.xAnyAlarm := dataBeltClean.AlSummary.xAlarmCritical OR dataBeltClean.AlSummary.xAlarmStop OR dataBeltClean.AlSummary.xAnyWarning;

	IF dataBeltClean.Commands.xReset THEN
		dataBeltClean.Alarm := ResetAlarms;
		dataBeltClean.AlSummary := ResetAlSummary;
	END_IF

	ars_AnyAlarm.xAlarm:= dataBeltClean.AlSummary.xAnyAlarm;
	ars_AnyAlarm.xSilence:=dataBeltClean.Commands.xMute;
	ars_AnyAlarm();

	dataBeltClean.AlSummary.xAlarmSound := ars_AnyAlarm.xAlarmSound;

END_ACTION
```

### Program Logical/ExtPack/_Transport/BeltCleaning/BeltCleaningSim/BeltCleaningSim (IEC)

#### BeltCleaningSim.st - Init, cyclic, exit code
```iecst
PROGRAM _INIT
	(* Insert code here *)
	BeltClean ACCESS ADR (gBeltClean);

	BeltClean.Inputs.xAirTurbVSDAvailable := TRUE;
	BeltClean.ParSw.tiCleaning := T#30s;
	BeltClean.ParSw.tiDrying := T#15s;

END_PROGRAM

PROGRAM _CYCLIC
	(* Insert code here *)
	IF BeltClean.Outputs.xAirTurbineVSDReset THEN
		BeltClean.Inputs.xAirTurbVSDAvailable := TRUE;
	END_IF
END_PROGRAM
```

### Program Logical/ExtPack/_Transport/BeltCtrl/BeltCtrl_v1/BeltCtrl (IEC)

#### BeltManager.st - Main is calling program actions
```iecst
PROGRAM _INIT

	//Define a transmision data to do the first calculations and be receptive to next calculations
	BeltDriveUnit.TransmissionData.TransmissionType := TRANS_LINEAL_PERIMETER;
	BeltDriveUnit.TransmissionData.LinealPerimeter.PulsesPerTurn := GC_UNITS_BY_REV_DRIVE;
	BeltDriveUnit.TransmissionData.LinealPerimeter.GearBox := 10.0;
	BeltDriveUnit.TransmissionData.LinealPerimeter.Perimeter := 500.0;

	//
	BeltDriveUnit.AccelerationDesired := 10;
	BeltDriveUnit.Calculation := CALC_ACC_PULSES;
	BeltDriveUnit();

	BeltDriveUnit.DecelerationDesired := 10;
	BeltDriveUnit.Calculation := CALC_DEC_PULSES;
	BeltDriveUnit();

END_PROGRAM

PROGRAM _CYCLIC

///////////////////////////////////////////////////////////////////////////////////////////////////////////////////////////////////////////////////////
// MAIN			MAIN			MAIN			MAIN			MAIN			MAIN			MAIN			MAIN			MAIN			MAIN
///////////////////////////////////////////////////////////////////////////////////////////////////////////////////////////////////////////////////////
// Main program is calling all program actions
///////////////////////////////////////////////////////////////////////////////////////////////////////////////////////////////////////////////////////

	// Reference AxisCtrl
	Belt ACCESS ADR (gBelt); //[RGP] This must point to an gBelt[iIndexBelt] in v2. FOR v1 stays as gBelt TO NOT modify the rest OF the PROGRAM were gBelt is being used
	AxisBelt ACCESS ADR (gAxis[Belt.parameters.IndexAxis]);

	// Reset action
	IF NOT Belt.parameters.xExistBelt THEN
		ResetAlarms;
		RETURN;
	END_IF

	// Reset Alarms
	IF Belt.commands.xReset THEN
		ResetAlarms;
	END_IF

	// Alarms action
	Alarms;

	// Critical alarms not allowing to do nothing
	IF Belt.Al.xAxisLengthNotDefined OR Belt.Al.xGearBoxNotDefined THEN
		RETURN;
	END_IF

	Belt.states.xOrderRuning := iBeltState=BELT_PREPARING_START OR iBeltState=BELT_RUN_ORDER OR iBeltState=BELT_RUNNING;

	///////////////////////////////////
	// In progress
	///////////////////////////////////

	BeltStates; // States Belt

	//Limits
	Belt.parameters.rSetPointSpeed := LIMIT(5.0, Belt.parameters.rSetPointSpeed, Belt.states.rMaxSpeed);
	IF Belt.parameters.xRemoteAcceleration AND Belt.commands.xUseJogAccDecc THEN
		Belt.states.rAcceleration := Belt.parSw.rAcceleration;
	ELSE
		Belt.states.rAcceleration := Belt.parameters.rAcceleration;
	END_IF
	Belt.states.rAcceleration := LIMIT(5.0, Belt.states.rAcceleration, Belt.parameters.rMaxAcceleration);

	IF Belt.parameters.xRemoteDeceleration AND Belt.commands.xUseJogAccDecc THEN
		Belt.states.rDeceleration := Belt.parSw.rDeceleration;

	ELSIF Belt.commands.xUseSoftDeceleration THEN
		Belt.states.rDeceleration := Belt.parameters.rSoftDeceleration;

	ELSE
		Belt.states.rDeceleration := Belt.parameters.rDeceleration;
	END_IF

	Belt.states.rDeceleration := LIMIT(500.0, Belt.states.rDeceleration, Belt.parameters.rMaxDeceleration);

	AxisBelt.Parameter.Direction:= Belt.parameters.Direction;

	xRunningState := iBeltState=BELT_RUNNING OR iBeltState=BELT_RUN_ORDER OR iBeltState=BELT_JOGGING;

	//Set velocity. Calculate speed in pulses with DriveUnit
	BeltDriveUnit.TransmissionData := Belt.parameters.DriveUnit;
	BeltDriveUnit.SpeedMminDesired := MAX(Belt.parameters.rSetPointSpeed, 0.5); 	//It avoids a 0 speed and do not see a Continuous Movement state
	BeltDriveUnit.Calculation := CALC_SPEED_MMIN_PULSES;
	BeltDriveUnit();

	//Definet the Status of the BELT with the Status of the Axis
	BeltDriveUnit.PulsesSpeedDevice := AxisBelt.Status.ActVelocity;
	BeltDriveUnit.Calculation := CALC_SPEED_MMIN;
	BeltDriveUnit();

	Belt.states.rCurrentSpeed	:= ABS(BeltDriveUnit.SpeedMminDevice);
	Belt.states.rCurrentSpeedUnits := ABS(AxisBelt.Status.ActVelocity);

	Belt.states.rMaxTemperature := ABS(AxisBelt.Status.MaxTempMotor);

	BeltDriveUnit.RevMinSpeedDevice := AxisBelt.Status.MaxSpeed;
	BeltDriveUnit.Calculation := CALC_SPEED_REVMIN_MMIN;
	BeltDriveUnit();
	Belt.states.Hw.rMaxSpeed := ABS(BeltDriveUnit.SpeedRpmToMmin);

	BeltDriveUnit.AccelerationDesired := Belt.states.rAcceleration;
	BeltDriveUnit.Calculation := CALC_ACC_PULSES;
	BeltDriveUnit();
	AxisBelt.Parameter.Acceleration := BeltDriveUnit.pulsesAccelerationDesired;

	BeltDriveUnit.DecelerationDesired := Belt.states.rDeceleration;
	BeltDriveUnit.Calculation := CALC_DEC_PULSES;
	BeltDriveUnit();
	AxisBelt.Parameter.Deceleration := BeltDriveUnit.pulsesDecelerationDesired;

	Belt.states.rActualCurrent := AxisBelt.Status.ActCurrent;

	Belt.states.rMaxTorque := ABS(MAX(AxisBelt.Status.MaxTorque, 0.001)); //rMaxTorque cannot be negative and cannot be 0

	IF Belt.states.rCurrentSpeed = 0 THEN
		Belt.states.rCurrentTorque	:= 0;
	ELSE
		Belt.states.rCurrentTorque	:= AxisBelt.Status.ActTorque;
	END_IF
	Belt.states.rCurrentTorque := ABS(Belt.states.rCurrentTorque);

	IF AxisBelt.Status.RatedTorque <> 0 THEN
		Belt.states.rTorquePerc		:= ABS(Belt.states.rCurrentTorque*100/AxisBelt.Status.RatedTorque);
	END_IF

	IF AxisBelt.Status.MaxAccelerationPos <> 0 THEN
		BeltDriveUnit.PulsesAccelerationDevice := AxisBelt.Status.MaxAccelerationPos;
		BeltDriveUnit.Calculation := CALC_ACC_MM;
		BeltDriveUnit();

		Belt.states.MaxPosAcceleration	:= ABS(BeltDriveUnit.mmAcceleration);
	END_IF

	IF AxisBelt.Status.MaxDecelerationPos <> 0 THEN
		BeltDriveUnit.PulsesDecelerationDevice := AxisBelt.Status.MaxDecelerationPos;
		BeltDriveUnit.Calculation := CALC_DEC_MM;
		BeltDriveUnit();

		Belt.states.MaxPosDeceleration	:= ABS(BeltDriveUnit.mmDeceleration);
	END_IF

	IF AxisBelt.Status.MaxAccelerationNeg <> 0 THEN
		BeltDriveUnit.PulsesAccelerationDevice := AxisBelt.Status.MaxAccelerationNeg;
		BeltDriveUnit.Calculation := CALC_ACC_MM;
		BeltDriveUnit();

		Belt.states.MaxNegAcceleration	:= ABS(BeltDriveUnit.mmAcceleration);
	END_IF

	IF AxisBelt.Status.MaxDecelerationNeg <> 0 THEN
		BeltDriveUnit.PulsesDecelerationDevice := AxisBelt.Status.MaxDecelerationNeg;
		BeltDriveUnit.Calculation := CALC_DEC_MM;
		BeltDriveUnit();

		Belt.states.MaxNegDeceleration	:= ABS(BeltDriveUnit.mmDeceleration);
	END_IF

	Belt.states.ErrorId 		:= AxisBelt.Status.ErrorID;

	//Just activating the signal with the order, so when stopping, the signal is lowered faster
	Belt.states.xRuningBelt		:= AxisBelt.Status.PLCopenState.ContinuousMotion AND (Belt.commands.xRunBelt OR Belt.commands.xJogBelt);

	//Calculation of belt's motor position
	BeltDriveUnit.pulsesDevice := AxisBelt.Status.ActPosition;
	BeltDriveUnit.Calculation := CALC_POS_MM;
	BeltDriveUnit();
	Belt.states.rMotorPosition := BeltDriveUnit.PositionDevice;

	// Sending axis motion orders
	AxisBelt.Command.Move.Halt     := AxisBelt.Status.PLCopenState.ContinuousMotion AND NOT xRunningState;
	AxisBelt.Command.Move.Velocity := EDGEPOS(xRunningState) OR (xRunningState AND AxisBelt.Parameter.Speed <> BeltDriveUnit.pulsesSpeedDesired); // JMH: It is important the order of these two lines
	AxisBelt.Parameter.Speed       := BeltDriveUnit.pulsesSpeedDesired; // JMH: It is important the order of these two lines

	Belt.states.rMaxSpeed := MIN(Belt.parameters.rMaxSpeed, Belt.states.Hw.rMaxSpeed);

	iTimesExecuted:=iTimesExecuted+1;

END_PROGRAM
```

#### AlarmsSummary.st - Belt alarms summary
```iecst
ACTION AlarmsSummary:

	//////////////////////////////
	//SUMMARY BELT ALARMS
	//////////////////////////////

	iReasonWarning.0 := Belt.Al.xBeltMotorTemp;
	iReasonWarning.1 := Belt.Al.xBeltDriverTemp;
	iReasonWarning.2 := Belt.Al.xWrnOverTorq;

	Belt.AlSummary.xAnyWarning:= iReasonWarning > 0;
	IF EDGEPOS(Belt.AlSummary.xAnyWarning) THEN
		Belt.AlSummary.iReasonWarning := iReasonWarning;
		LogWarning;
	ELSIF EDGEPOS(NOT Belt.commands.AutoMode.xStop AND NOT Belt.AlSummary.xAlarmStop) THEN
		Belt.AlSummary.iReasonWarning := 0;
	END_IF

	// Stop alarms are drive alarms but just when are not from safety
	iReasonStop.0 := Belt.Al.xAnyDriveAlarm;
	iReasonStop.1 := Belt.Al.xAlrComDrive;
	iReasonStop.2 := Belt.Al.xAlrPowerBeltError;
	iReasonStop.3 := Belt.Al.xAlrProtDrive;
	iReasonStop.4 := Belt.Al.xAlrOverTorque;
	iReasonStop.5 := Belt.Al.xControllerNotReady;
	iReasonStop.6 := Belt.Al.xEnableVoltageSag;

	Belt.AlSummary.xAlarmStop:=	iReasonStop > 0;
	IF EDGEPOS(Belt.AlSummary.xAlarmStop) THEN
		Belt.AlSummary.iReasonStop[0] := iReasonStop;
		LogStopAlarm;
	ELSIF EDGEPOS(NOT Belt.commands.AutoMode.xStop AND NOT Belt.AlSummary.xAlarmStop) THEN
		Belt.AlSummary.iReasonStop[0] := 0;
	END_IF

	// Summary Alarms (Critical, Sound, Warnings, Stop )
	iReasonCritical.1 := Belt.Al.xAxisLengthNotDefined;
	iReasonCritical.1 := Belt.Al.xGearBoxNotDefined;

	Belt.AlSummary.xAlarmCritical:= iReasonCritical>0;
	//Register the reason of the Critical Alarm
	IF Belt.commands.Mode.xAuto AND EDGEPOS(Belt.AlSummary.xAlarmCritical) THEN
		Belt.AlSummary.iReasonCritical := iReasonCritical;
		LogCriticalAlarm;
	ELSIF EDGEPOS(Belt.commands.Mode.xAuto AND NOT Belt.AlSummary.xAlarmCritical) THEN
		Belt.AlSummary.iReasonCritical := 0;
	END_IF

	Belt.AlSummary.xAlrSafetySystemGeneral := Belt.commands.xExternalSafetyStop;

	Belt.AlSummary.xAnyAlarm:= Belt.AlSummary.xAlarmCritical OR Belt.AlSummary.xAlarmStop OR Belt.AlSummary.xAlrSafetySystemGeneral;

	// Alarms reseteable sound management.
	ars_AlrStop.xAlarm:= Belt.AlSummary.xAlarmStop;
	ars_AlrStop.xSilence:= Belt.commands.xMute;
	ars_AlrStop();

	ars_AlrCritical.xAlarm:= Belt.AlSummary.xAlarmCritical;
	ars_AlrCritical.xSilence:= Belt.commands.xMute;
	ars_AlrCritical();

	ars_AlrWarning.xAlarm:= Belt.AlSummary.xAnyWarning;
	ars_AlrWarning.xSilence:= Belt.commands.xMute;
	ars_AlrWarning();

	Belt.AlSummary.xAlarmSound:= 	//ars_AlrWarning.xAlarmSound OR
									ars_AlrStop.xAlarmSound OR
									ars_AlrCritical.xAlarmSound;

END_ACTION
```

#### BeltStates.st - Belt states control
```iecst
ACTION BeltStates:

	// ####################################################################
	// ####################################################################
	//
	// Check BeltStates.graphml to understand better this implementation

	// Here will be implemented a belt states controller,
CASE iBeltState OF

	BELT_NOT_INITIALIZED:
		// PowerOn Command
		IF AxisBelt.Status.ControllerReady AND NOT Belt.commands.Mode.xZero THEN
			// Switched on
			AxisBelt.Command.Power:=TRUE;
			iBeltState:=BELT_SWITCH_ON;
			AxisBelt.Command.ErrorAcknowledge:= TRUE;

		END_IF
		ResetKnownSafetyErrors;

	BELT_SWITCH_ON:

		IF (NOT AxisBelt.Status.HomeOK) AND AxisBelt.Status.PowerOn THEN
			//Doing Home Direct
			iBeltState:=BELT_HOMING;
			AxisBelt.Command.HomeDirect :=TRUE;
		ELSIF AxisBelt.Status.HomeOK THEN
			// All is initialized
	    	iBeltState:=BELT_INITIALIZED;
		END_IF;

	BELT_HOMING:
		IF AxisBelt.Status.HomeOK THEN
			//Doneg Home Direct
			iBeltState:=BELT_INITIALIZED;
		END_IF

	BELT_INITIALIZED:
		// Belt is initialized when axis state is StandStill
		// Waiting for enabled to run state
		IF AxisBelt.Status.PLCopenState.StandStill THEN
			// Ready for movements
			iBeltState:=BELT_IDLE;
		ELSIF AxisBelt.Status.PLCopenState.ErrorStop OR AxisBelt.Status.PLCopenState.Disabled THEN
			// Some was wrong!!!
			iBeltState:=BELT_ERROR;
		END_IF

	BELT_IDLE:
		// Waiting for movements
		// Command start belt movement
		IF Belt.commands.xRunBelt THEN
			iBeltState:=BELT_PREPARING_START;
		END_IF

		IF Belt.commands.xJogBelt THEN
			iBeltState:=BELT_JOGGING;
		END_IF

	BELT_PREPARING_START:
		IF NOT Belt.commands.xRunBelt THEN
			iBeltState:=BELT_IDLE;

		ELSIF (Belt.commands.Mode.xAuto) AND NOT Belt.commands.xConsentBelt THEN
			// Waiting for consent
			iBeltState:=BELT_NOT_CONSENT;

		ELSIF xRunBeltOrderAfterSound THEN
			// Waiting for movements
			iBeltState:=BELT_RUN_ORDER;
		END_IF

	BELT_RUN_ORDER:
		//Launched movement
		IF NOT Belt.commands.xRunBelt THEN
			iBeltState:=BELT_IDLE;

		ELSIF (Belt.commands.Mode.xAuto) AND NOT Belt.commands.xConsentBelt THEN
			// Waiting for consent
			iBeltState:=BELT_NOT_CONSENT;

		ELSIF Belt.states.xRuningBelt THEN
			// Waiting for movements
			iBeltState:=BELT_RUNNING;
		END_IF

	BELT_RUNNING:
		IF NOT Belt.commands.xRunBelt THEN
			iBeltState:=BELT_IDLE;

		ELSIF (Belt.commands.Mode.xAuto) AND NOT Belt.commands.xConsentBelt THEN
			// Waiting for consent
			iBeltState:=BELT_NOT_CONSENT;
		END_IF

	BELT_JOGGING:
		IF NOT Belt.commands.xJogBelt THEN
			iBeltState:=BELT_IDLE;
		END_IF

	BELT_NOT_CONSENT:
		IF NOT Belt.commands.xRunBelt THEN
			iBeltState:=BELT_IDLE;

		ELSIF Belt.commands.xConsentBelt THEN
			// Consent received
			iBeltState:=BELT_PREPARING_START;
		END_IF

	BELT_ERROR:

		iTimesExecutedErrorState:=iTimesExecutedErrorState+1;

		// Reset & ERRROR MANAGEMENT
		//
		// Power off
		AxisBelt.Command.Power:=FALSE;

		// Manual recovery:
		AxisBelt.Command.Reset:= (NOT AxisBelt.Status.ControllerReady AND Belt.commands.xReset); // OR
								//tpResetAnyDriveAlarm.Q;

		// Auto reseteable Id code as fast recovery:
		// Error Id 6023: Voltage sag at controller enable input
		// Error If 29209: MC_Power
		// Error if 29207: MC_Home
		// Error if 29206: MC_MoveVelocity ? gives this error because controller is off
		// Error if 29216: MC_MoveVelocity ? gives this error because continuous movement is not possible
		// Error if 29217: Invalid input parameter

		ResetKnownSafetyErrors;

		//TOREVIEW: Why just acknowledge "known" errors????
		//TOREMOVE: AxisBelt.Command.ErrorAcknowledge:=(AxisBelt.Status.ErrorID = 29209) OR (AxisBelt.Status.ErrorID = 29207);
		AxisBelt.Command.ErrorAcknowledge:= Belt.commands.xReset;

		IF NOT Belt.Al.xAnyDriveAlarm THEN
			iBeltState:= BELT_NOT_INITIALIZED;
		END_IF

	END_CASE

	/////////////////////////////////
	// Update belt states
	/////////////////////////////////

	// xZero state changes Belt state to not initialized
	// It avoids transport belt errors
	IF (Belt.commands.Mode.xZero) THEN
		iBeltState:=BELT_NOT_INITIALIZED;
		// Error state changes Belt state
	ELSIF Belt.Al.xAnyDriveAlarm THEN
		iBeltState:=BELT_ERROR;
	END_IF

	//Saving state history
	IF iBeltState<>StateHistory[0] THEN
		FOR iIndexHistory:=iHistoryLines TO 1 BY -1 DO
			StateHistory[iIndexHistory]:=StateHistory[iIndexHistory-1];
		END_FOR
		StateHistory[0]:=iBeltState;
	END_IF

	Belt.states.State:=	iBeltState;

	///////////////////////
	// Timer management
	///////////////////////

	// Timer sounds Belt starting
	T_SoundBelt.IN:= iBeltState=BELT_PREPARING_START;
	// If time beeping not configured, use default value
	IF Belt.parameters.tiTimeBeepBeforeMove = 0 THEN
		T_SoundBelt.PT:= T#3s;
	ELSE
		T_SoundBelt.PT:= Belt.parameters.tiTimeBeepBeforeMove;
	END_IF
	T_SoundBelt();
	xRunBeltOrderAfterSound:=T_SoundBelt.Q;

	//Pulse to set a command reset to drive when in error state
	tpResetAnyDriveAlarm(IN:=Belt.Al.xAnyDriveAlarm, PT:=T#500ms);

END_ACTION

ACTION ResetKnownSafetyErrors:

	IF xAvoidResettingSafetyErrors THEN
		RETURN;
	END_IF

	iReasonAutoAcknowledge.0 := AxisBelt.Status.ErrorID = 29209;
	iReasonAutoAcknowledge.1 := AxisBelt.Status.ErrorID = 6058; // Not signal in Enable 1
	iReasonAutoAcknowledge.2 := AxisBelt.Status.ErrorID = 6059; // Not signal in Enable 2
	iReasonAutoAcknowledge.3 := AxisBelt.Status.ErrorID = 6023;
	iReasonAutoAcknowledge.4 := AxisBelt.Status.ErrorID = 4005;
	iReasonAutoAcknowledge.5 := AxisBelt.Status.ErrorID = 29203; //Not possible to start controller

	// If the drive has Enable errors but we know we have a Safety problem, auto acknowledge the errors
	IF (*Belt.commands.xExternalSafetyStop AND*) iReasonAutoAcknowledge > 0 THEN
		AxisBelt.Command.ErrorAcknowledge := TRUE;
	END_IF

END_ACTION
```

### Program Logical/ExtPack/_Transport/EdgeHoldDown/EdgeHoldDown_v1/EdgeHoldDown (IEC)

#### EdgeHoldDown.var
```iecst
VAR
	data : REFERENCE TO EdgeHoldDown_typ;
	AdjustmentSystem : REFERENCE TO ARRAY[0..2] OF PairedIclaMotors_typ;
	stAlarmsReseted : EdgeHoldDownAlarms;
	stEhdAlarmSummaryReseted : stEFI_AlarmSummary;
	rSensorPositionAlignment : REAL; (*Pulses*)
	rSensorPositionAlignmentMax : REAL; (*Pulses*)
	rSensorPositionAlignmentMin : REAL; (*Pulses*)
	rSensorPositionDesired : REAL; (*Pulses*)
END_VAR
VAR CONSTANT
	iHistoryLines : USINT := 20;
END_VAR
VAR
	tonMaxTimeJogging : TON;
	xAnyManualMovement : BOOL;
	rPositionMotorMm : REAL;
	ars_AlrStop : AutoResetSound;
	ars_AlrCritical : AutoResetSound;
	ars_AlrWarning : AutoResetSound;
	ResetCommands : EdgeHoldDownCommands;
	iCancelMovement : USINT;
	iReasonWarning : UDINT;
	iReasonStop : UDINT;
	iReasonCritical : UDINT;
	StateHistory : ARRAY[0..iHistoryLines] OF EdgeHoldDownState;
	iIndexHistory : USINT;
	MotorDriveUnit : DriveUnitMngr;
	rJogSpeedSetPoint : REAL;
	xControllerReady : BOOL;
	xPoweredOn : BOOL;
	xMotorReady : BOOL;
	xAnyError : BOOL;
	xAnyManualOrder : BOOL;
	iIndexSensor : USINT;
	iAnyWarning : UINT;
	tonMotorStopped : TON;
	xMotorStopped : BOOL;
	stCriticalAlarmsLog : EventLog_typ;
	stStopAlarmsLog : EventLog_typ;
	stWarningAlarmsLog : EventLog_typ;
	iIndexIclaMotor : USINT;
	iIndexAdjustmentSystem : USINT;
	iCancelHoming : USINT;
	iPositionState : EdgeHoldDownPositionStates;
	rWidthAdjustPosition : REAL;
	rHeighAdjustPosition : REAL;
	iSystemState : EdgeHoldDownState;
	iSystemAutoState : EdgeHoldDownAutoState;
	iNumIclaMotors : USINT;
	iMisalignmentToleranceInAuto : USINT := 5;
	iMisalignmentToleranceInManual : USINT := 10;
	iSafetyOffset : USINT := 5;
	ResetCommandsSw : EdgeHoldDownCommandsSw;
END_VAR
```

#### Configuration.st
```iecst
ACTION Configuration:

	data.status.EdgeHoldDownType := EHDTY_V2;

	//Case not used currently because the only type used by platforms based in OnePlc (B&R) is V2 type.
	//This type assignation is required BY SW team TO manage their UI

//	CASE data.status.EdgeHoldDownType OF
//		EHDTY_V1:
//
//
//		EHDTY_V2:
//
//
//	END_CASE

END_ACTION
```

#### MachineState.st
```iecst
ACTION MachineState:

	data.parameters.rBarsOffset := LIMIT(data.Hw.iMinBarsOffset, data.parSw.rBarsOffset, data.Hw.iMaxBarsOffset);
	rHeighAdjustPosition := (data.parameters.rBarsHeighSp + data.parameters.rBarsOffset);
	rWidthAdjustPosition := (data.parameters.rWidthSp - data.parSw.iOverlap*2); //Multiplied by two so overlap refers to each metal band/strap
	rWidthAdjustPosition := (rWidthAdjustPosition-data.Hw.rMinWidthAdjustment)/2;

	//Saving ski position
	data.status.rSkiPosition := AdjustmentSystem[1].Motor[1].rPositionMotor - data.parameters.rDistanceMetalBandToSki;

	data.status.rBlockPrePrintingPosition := rHeighAdjustPosition*2; //Setting a big margin to avoid to damage printheads when moving ehd metal bands

	CheckMotorsInPosition;
	CheckMotorsInRestingPosition;
	CheckMotorsInAdjustedPosition;

	CASE iSystemState OF
		EHD_STOPPED:
			ResetSwOrders;

			//Resetting orders (zero state)
			data.orders.xAdjustToMedia:=FALSE;
			data.orders.xResetPosition:=FALSE;

			//Manual mode
			IF (data.commands.Mode.xManual) THEN
				iSystemState:=EHD_MANUAL;

			//Auto
			ELSIF data.commands.Mode.xAuto AND data.status.xReferenced THEN
				iSystemState:=EHD_IDLE;
			END_IF

		EHD_MANUAL:
			//Setting parameters that depend on ehd mode
			AdjustmentSystem[1].parameters.iMisalignmentTolerance := iMisalignmentToleranceInManual;
			AdjustmentSystem[2].parameters.iMisalignmentTolerance := iMisalignmentToleranceInManual;

			//Logic ctrl
			ManualLogic;

		EHD_IDLE:
			//Setting parameters that depend on ehd mode
			AdjustmentSystem[1].parameters.iMisalignmentTolerance := iMisalignmentToleranceInAuto;
			AdjustmentSystem[2].parameters.iMisalignmentTolerance := iMisalignmentToleranceInAuto;

			//Logic ctrl
			AutoLogic;

		EHD_ERROR:
			ResetSwOrders;
			IF NOT xAnyError THEN
				iSystemState := EHD_STOPPED;
			END_IF
	END_CASE

	IF NOT data.parameters.xEnableMovements OR (iSystemState=EHD_STOPPED) THEN
		AdjustmentSystem[1].parameters.xMovementsEnabled := FALSE;
		AdjustmentSystem[2].parameters.xMovementsEnabled := FALSE;

	//In automatic enable depends on motor positions
	ELSIF (iSystemState=EHD_IDLE) THEN

															//Enable in case metal bands are not high enough to damage photocells chassis
		AdjustmentSystem[1].parameters.xMovementsEnabled :=	(AdjustmentSystem[1].Motor[1].rPositionMotor <= (data.Hw.rMaxDistanceMetalBandToBelt - iSafetyOffset)) OR
															//Enable movements in case where metal bands are not below photocells lasers
															(AdjustmentSystem[2].Motor[1].rPositionMotor <= gMachine.Pt.Hw.iWidth);

		AdjustmentSystem[2].parameters.xMovementsEnabled := (data.status.rSkiPosition >= (iSafetyOffset - AdjustmentSystem[2].Motor[1].rMotorResolution));

	ELSE

		AdjustmentSystem[1].parameters.xMovementsEnabled := TRUE;
		AdjustmentSystem[2].parameters.xMovementsEnabled := TRUE;
	END_IF

	//In Zero mode it goes to not Init
	IF (data.commands.Mode.xZero) THEN
		iSystemState:=EHD_STOPPED;

	ELSIF xAnyError THEN
		iSystemState:=EHD_ERROR;
	END_IF

	//Saving state history
	IF iSystemState<>StateHistory[0] THEN
		FOR iIndexHistory:=iHistoryLines TO 1 BY -1 DO
			StateHistory[iIndexHistory]:=StateHistory[iIndexHistory-1];
		END_FOR
		StateHistory[0]:=iSystemState;
	END_IF

	//AutoLogic ctrl
	IF iSystemState<>EHD_IDLE THEN
		iSystemAutoState := EHD_OUT_OF_AUTO;
	END_IF

	//State summary
	data.status.iSystemState:=iSystemState;
	data.status.xMoving := AdjustmentSystem[1].status.xMoving OR AdjustmentSystem[2].status.xMoving;
	data.status.xReferenced := AdjustmentSystem[1].status.xReferenced AND AdjustmentSystem[2].status.xReferenced;
	data.status.xReferencing := AdjustmentSystem[1].status.xReferencing OR AdjustmentSystem[2].status.xReferencing;
	data.status.xReady := data.parameters.xEnableMovements AND data.status.xEnabled;
	data.status.xAdjusting := (iSystemAutoState = EHD_ADJUSTING_STEP_1) OR (iSystemAutoState = EHD_ADJUSTING_STEP_2) OR (iSystemAutoState = EHD_ADJUSTING_STEP_3);
	data.status.xGoingRestPosition := (iSystemAutoState = EHD_RESTING_STEP_1) OR (iSystemAutoState = EHD_RESTING_STEP_2) OR (iSystemAutoState = EHD_RESTING_STEP_3);

	data.commands.xStop := FALSE;

END_ACTION

ACTION ManualLogic:
	IF data.parameters.xEnableMovements THEN
		//Commands
		//Reference systems
		AdjustmentSystem[1].commands.xReference:= data.commandsSw.xReference;
		AdjustmentSystem[2].commands.xReference:= data.commandsSw.xReference;

		//Movements
		IF NOT AdjustmentSystem[1].status.xReferencing AND NOT AdjustmentSystem[1].commands.xReference THEN
			AdjustmentSystem[1].commands.xMoveBackward := data.ordersSw.xMoveUp;
			AdjustmentSystem[1].commands.xMoveForward := data.ordersSw.xMoveDown;
		END_IF

		IF NOT AdjustmentSystem[2].status.xReferencing AND NOT AdjustmentSystem[2].commands.xReference THEN
			AdjustmentSystem[2].commands.xMoveBackward := data.ordersSw.xMoveBackward; //To move metal bands to the edge of the belt
			AdjustmentSystem[2].commands.xMoveForward := data.ordersSw.xMoveForward; //To move metal bands to the center of the belt
		END_IF

		//Alarm excessive manual commands activated
		tonMaxTimeJogging.IN:= 	(data.ordersSw.xMoveBackward OR
								data.ordersSw.xMoveForward OR
								data.ordersSw.xMoveDown OR
								data.ordersSw.xMoveUp);
		tonMaxTimeJogging.PT:= T#5S;
		tonMaxTimeJogging();

		// Stopping all
		IF tonMaxTimeJogging.Q THEN
			ResetSwOrders;
		END_IF
	END_IF

	IF data.status.xReferencing THEN
		data.commandsSw.xReference := FALSE;
	END_IF

END_ACTION

ACTION AutoLogic:

	CASE iSystemAutoState OF

		EHD_OUT_OF_AUTO:
			iSystemAutoState := EHD_MOVEMENTS_NOT_ENABLED;

		EHD_MOVEMENTS_NOT_ENABLED:
			AdjustmentSystem[1].commands.xStop := TRUE;
			AdjustmentSystem[2].commands.xStop := TRUE;
			IF data.parameters.xEnableMovements THEN
				iSystemAutoState := EHD_READY;
			END_IF

		EHD_READY:
			//To review how to reset these commands using an action instead of assigning FALSE here.
			AdjustmentSystem[1].commands.xStop := FALSE;
			AdjustmentSystem[2].commands.xStop := FALSE;
			IF (EDGEPOS(data.orders.xResetPosition) OR NOT data.parSw.xEnable) AND NOT data.status.xInRestingPosition THEN
				AdjustmentSystem[1].parameters.rPositionDesired := data.parameters.rDistanceMetalBandToSki + iSafetyOffset;
				iSystemAutoState := EHD_RESTING_STEP_1;

			ELSIF EDGEPOS(data.orders.xAdjustToMedia) AND NOT data.status.xAdjustedToMedia THEN
				IF AdjustmentSystem[2].parameters.rPositionDesired <> rWidthAdjustPosition THEN
					//Assigning resting position as desired position to move metal bands in cross direction
					AdjustmentSystem[1].parameters.rPositionDesired := data.parameters.rDistanceMetalBandToSki + iSafetyOffset;
					iSystemAutoState := EHD_ADJUSTING_STEP_1;
				ELSE
					//Going to state where desired heigh position is set as desired position to move metal bands in vertical direction
					iSystemAutoState := EHD_ADJUSTING_STEP_2;
				END_IF
			END_IF

		EHD_ADJUSTING_STEP_1:
			//Moving system up. Waiting to arrive to desired position
			IF AdjustmentSystem[1].status.xInPosition THEN
				AdjustmentSystem[2].parameters.rPositionDesired := rWidthAdjustPosition;
				iSystemAutoState := EHD_ADJUSTING_STEP_2;
			END_IF

		EHD_ADJUSTING_STEP_2:
			//Moving system to widht adjust position. Waiting to arrive to desired position
			IF AdjustmentSystem[2].status.xInPosition THEN
				AdjustmentSystem[1].parameters.rPositionDesired := rHeighAdjustPosition;
				iSystemAutoState := EHD_ADJUSTING_STEP_3;
			END_IF

		EHD_ADJUSTING_STEP_3:
			//Moving up system to height adjust position. Waiting to arrive to desired position
			IF AdjustmentSystem[1].status.xInPosition THEN
				iSystemAutoState := EHD_READY;
			END_IF

		EHD_RESTING_STEP_1:
			//Moving system down. Waiting to arrive to desired position
			IF AdjustmentSystem[1].status.xInPosition THEN
				AdjustmentSystem[2].parameters.rPositionDesired := AdjustmentSystem[2].parameters.rMechPositionMax;
				iSystemAutoState := EHD_RESTING_STEP_2;
			END_IF

		EHD_RESTING_STEP_2:
			//Moving system to width resting position. Waiting to arrive to desired position
			IF AdjustmentSystem[2].status.xInPosition THEN
				AdjustmentSystem[1].parameters.rPositionDesired := AdjustmentSystem[1].parameters.rMechPositionMin;
				iSystemAutoState := EHD_RESTING_STEP_3;
			END_IF

		EHD_RESTING_STEP_3:
			//Moving system to height resting position. Waiting to arrive to desired position
			IF AdjustmentSystem[1].status.xInPosition THEN
				iSystemAutoState := EHD_READY;
			END_IF

	END_CASE

	AdjustmentSystem[1].parameters.rPositionDesired := LIMIT(AdjustmentSystem[1].parameters.rMechPositionMin,AdjustmentSystem[1].parameters.rPositionDesired, AdjustmentSystem[1].parameters.rMechPositionMax);
	AdjustmentSystem[2].parameters.rPositionDesired := LIMIT(AdjustmentSystem[2].parameters.rMechPositionMin,AdjustmentSystem[2].parameters.rPositionDesired, AdjustmentSystem[2].parameters.rMechPositionMax);

	//To stop process taking place when any stop alarm is raised
	iCancelMovement.0 := data.AlSummary.xAlarmStop;
	iCancelMovement.1 := data.commands.xStop;
	iCancelMovement.2 := NOT data.parameters.xEnableMovements;

	IF iCancelMovement>0 THEN
		iSystemAutoState := EHD_MOVEMENTS_NOT_ENABLED;
	END_IF

END_ACTION

ACTION CheckMotorsInPosition:

	data.status.xInPosition := (ABS(AdjustmentSystem[1].parameters.rPositionDesired-AdjustmentSystem[1].Motor[1].rPositionMotor)<AdjustmentSystem[1].Motor[1].rMotorResolution) AND
								(ABS(AdjustmentSystem[1].parameters.rPositionDesired-AdjustmentSystem[1].Motor[2].rPositionMotor)<AdjustmentSystem[1].Motor[2].rMotorResolution) AND
								(ABS(AdjustmentSystem[2].parameters.rPositionDesired-AdjustmentSystem[2].Motor[1].rPositionMotor)<AdjustmentSystem[2].Motor[1].rMotorResolution) AND
								(ABS(AdjustmentSystem[2].parameters.rPositionDesired-AdjustmentSystem[2].Motor[2].rPositionMotor)<AdjustmentSystem[2].Motor[2].rMotorResolution);
END_ACTION

ACTION CheckMotorsInAdjustedPosition:

	data.status.xAdjustedToMedia := (ABS(rHeighAdjustPosition-AdjustmentSystem[1].Motor[1].rPositionMotor)<AdjustmentSystem[1].Motor[1].rMotorResolution) AND
									(ABS(rHeighAdjustPosition-AdjustmentSystem[1].Motor[2].rPositionMotor)<AdjustmentSystem[1].Motor[2].rMotorResolution) AND
									(ABS(rWidthAdjustPosition-AdjustmentSystem[2].Motor[1].rPositionMotor)<AdjustmentSystem[2].Motor[1].rMotorResolution) AND
									(ABS(rWidthAdjustPosition-AdjustmentSystem[2].Motor[2].rPositionMotor)<AdjustmentSystem[2].Motor[2].rMotorResolution);
END_ACTION

ACTION CheckMotorsInRestingPosition:

	data.status.xInRestingPosition := (ABS(AdjustmentSystem[1].parameters.rMechPositionMin-AdjustmentSystem[1].Motor[1].rPositionMotor)<AdjustmentSystem[1].Motor[1].rMotorResolution) AND
										(ABS(AdjustmentSystem[1].parameters.rMechPositionMin-AdjustmentSystem[1].Motor[2].rPositionMotor)<AdjustmentSystem[1].Motor[2].rMotorResolution) AND
										(ABS(AdjustmentSystem[2].parameters.rMechPositionMax-AdjustmentSystem[2].Motor[1].rPositionMotor)<AdjustmentSystem[2].Motor[1].rMotorResolution) AND
										(ABS(AdjustmentSystem[2].parameters.rMechPositionMax-AdjustmentSystem[2].Motor[2].rPositionMotor)<AdjustmentSystem[2].Motor[2].rMotorResolution);
END_ACTION
```

#### ResetCommands.st
```iecst
ACTION ResetSwOrders:
	data.ordersSw.xMoveUp    := FALSE;
	data.ordersSw.xMoveDown  := FALSE;
	data.ordersSw.xMoveBackward := FALSE;
	data.ordersSw.xMoveForward := FALSE;
END_ACTION
```

### DocEhd.md
```markdown
| Doc Version | Description   | Date       | Resp     |
| ----------- | ------------- | ---------- | -------- |
| 1.0         | First release | 15/05/2024 | R.Gallén |
|             |               |            |          |
|             |               |            |          |

# Related documentation

[Lexium Integrated Drive Product manual](https://efi365.sharepoint.com/:b:/r/sites/inkjet/cretaprint/oficinatecnica2/Lean%20Product%20Development/Controls/05%20Interesting%20data/ILE/ILE1B_ILE1F_ILE1R_manual_V200_logo-EN.pdf?csf=1&web=1&e=0NQaF1)

[[20220803_EHD_NZ2_DESIGN REVIEW.pptx](https://efi365.sharepoint.com/:p:/r/sites/inkjet/cretaprint/proyectos/DeLorean/Shared%20Documents/02%20R%26D,%20APP/00%20Concept/Stage2/20220803_EHD_NZ2_DESIGN%20REVIEW.pptx?d=w27b4d2092bb34d2cac40ef445c414003&csf=1&web=1&e=OYqolg)](https://efi365.sharepoint.com/:p:/r/sites/inkjet/cretaprint/proyectos/DeLorean/Shared%20Documents/02%20R%26D,%20APP/00%20Concept/Stage2/EHD_NZ2_SW_PLC_DESIGN%20REVIEW.pptx?d=w4ccdfc3dd7c74b43848b5da3ef0d8387&csf=1&web=1&e=zBDZgC)

# How to use the package

***Commands***:

| Name     | Type                   | Description                                     |
| -------- | ---------------------- | ----------------------------------------------- |
| AutoMode | stEFI_MachineAutoModes | Starts a movement in the positive direction     |
| Mode     | StGeneral_States_Mode  | Machine general modes (manual, zero, automatic) |
| Mute     | BOOL                   | Mute active alarms sound                        |
| Reset    | BOOL                   | Acknowledges and quits all errors               |
| Stop     | BOOL                   |                                                 |

**CommandsSw**:

| Name      | Type | Description                 |
| --------- | ---- | --------------------------- |
| Reference | BOOL | Sets motors homing position |

**Orders**:

| Name          | Type | Description                                                                      |
| ------------- | ---- | -------------------------------------------------------------------------------- |
| ResetPosition | BOOL | Sets resting position (metal bands on the edge of the belt) as setpoint position |
| AdjustToMedia | BOOL | Sets adjusting position (metal bands overlapping board) as setpoint position     |

**OrdersSw**:

| Name         | Type | Description                                   |
| ------------ | ---- | --------------------------------------------- |
| MoveForward  | BOOL | To move metal bands to the center of the belt |
| MoveBackward | BOOL | To move metal bands to the edge of the belt   |
| MoveUp       | BOOL | To move metal bands up                        |
| MoveDown     | BOOL | To move metal bands down                      |

**Parameters**

| Name                    | Type  | Description                                                                                      |
| ----------------------- | ----- | ------------------------------------------------------------------------------------------------ |
| Installed               | BOOL  | Physical hardware related to ehd is installed                                                    |
| EnableMovements         | BOOL  | Ehd is enabled to perform movements                                                              |
| DistanceMetalBandToSki  | REAL  | Distance (in vertical) between ski and metal band (mm)                                           |
| WidthSp                 | REAL  | Metal bands width position setpoint (mm)                                                         |
| BarsOffset              | REAL  | Offset desired between metal bands height and bars position (mm)                                 |
| BarsHeighSp             | REAL  | Bars desired printing position (mm)                                                              |
| BlockPosition           | REAL  | Bars actual position (mm)                                                                        |
| AdjustmentSystemsNumber | USINT | Number of adjustment systems used by the edge hold down. Adjust system is composed by two motors |

**Hw Parameters**

| Name                       | Type | Description                                                                                                                 |
| -------------------------- | ---- | --------------------------------------------------------------------------------------------------------------------------- |
| iMinBarsOffset             | BOOL | Minimum bars offset allowed (mm)                                                                                            |
| iMaxBarsOffset             | BOOL | Maximum bars offsetallowed (mm)                                                                                             |
| iMinOverlap                | REAL | Minimum overlap allowed (mm)                                                                                                |
| iMaxOverlap                | REAL | Maximum overlap allowed (mm)                                                                                                |
| MinWidhtAdjustment         | REAL | Distance between sliders when inductive sensor for minimum position is active (mm)                                          |
| MaxDistanceMetalBandToBelt | REAL | Limited height where ehd can be moved vertically when postioned wider than belt's widht to avoid crash with 6l chassis (mm) |

**ParSw**

| Name        | Type | Description                                                      |
| ----------- | ---- | ---------------------------------------------------------------- |
| rBarsOffset | REAL | Offset desired between metal bands height and bars position (mm) |
| iOverlap    | UINT | Overlap between metal bands and media (mm)                       |
| xEnable     | BOOL | Activated via user interface                                     |

**Status**:

| Name                     | Type | Description                                                                                                                                         |
| ------------------------ | ---- | --------------------------------------------------------------------------------------------------------------------------------------------------- |
| BlockPrePrintingPosition | REAL | Desired block position calculated depending on metal bands position                                                                                 |
| Installed                | BOOL | Physical hardware related to ehd is installed and acknowledged                                                                                      |
| Enabled                  | BOOL | Ehd object is enabled                                                                                                                               |
| Referencing              | BOOL | Referencing process is taking place                                                                                                                 |
| Referenced               | BOOL | All motors required by ehd are referenced                                                                                                           |
| InRestingPosition        | BOOL | All adjustment systems are positioned at resting position                                                                                           |
| AdjustedToMedia          | BOOL | All adjustment systems are positioned at adjusting position                                                                                         |
| Moving                   | BOOL | Any adjustment system is moving                                                                                                                     |
| Ready                    | BOOL | All adjustment system are ready to operate (no errors)                                                                                              |
| InPosition               | BOOL | All adjustment systems are positioned at desired position (this variable is always active when "InRestingPosition" or "AdjustedToMedia" are active) |
| SkiPosition              | REAL | Position of ski (heigh) in mm                                                                                                                       |
| GoingRestPosition        | BOOL | Any adjustment system is moving to resting position                                                                                                 |
| Adjusting                | BOOL | Any adjustment system is moving to adjusting position                                                                                               |

**Inputs**:

| Name | Type | Description              |
| ---- | ---- | ------------------------ |
| Jam  | BOOL | Active when jam detected |

**Alarms**

| Name                 | Type | Description                                                                       |
| -------------------- | ---- | --------------------------------------------------------------------------------- |
| ParametersOutOfRange | REAL | Active when order to adjust media received and parameters are out of requirements |
| MovementsNotEnabled  | BOOL | Active when order to adjust to media received when movements are not enabled      |
| Jam                  | BOOL | Jam sensor has detect media while ehd is adjusted to media                        |
| NotReferenced        | BOOL | Any adjustment system not referenced                                              |

# State diagram

[Machine State diagram](EdgeHoldDown.graphml)

| State   | Action                                                     | Transition                                                                        |
| ------- | ---------------------------------------------------------- | --------------------------------------------------------------------------------- |
| ERROR   | REAL                                                       | Active when order to adjust media received and parameters are out of requirements |
| STOPPED | BOOL                                                       | Zero or Not Errors                                                                |
| MANUAL  | Receptive to reference command and manual movements orders | Machine in manual mode                                                            |
| AUTO    | Auto logic executed (see AutoState table)                  | Machine in automatic mode                                                         |

| AutoState                 | Action                                                          | Transition                                                         |
| ------------------------- | --------------------------------------------------------------- | ------------------------------------------------------------------ |
| EHD_OUT_OF_AUTO           | No action executed                                              | Machine not in auto state                                          |
| EHD_MOVEMENTS_NOT_ENABLED | Stop commands sent to paired motors                             | Movements are not enabled. Stop command received. AlarmStop active |
| EHD_READY                 | Stop commands released. Sets height adjustment system position. | Movements are enabled. Adjustment systems are positioned.          |
| EHD_RESTING_STEP_1        | Sets width adjustment system position.                          | ~~"ResetPosition" order received~~                                 |
| EHD_RESTING_STEP_2        | Sets height adjustment system position.                         | Height adjustment system is positioned                             |
| EHD_RESTING_STEP_3        | No action executed                                              | Width adjustment system is positioned                              |
| EHD_ADJUSTING_STEP_1      | Sets width adjustment system position.                          | "AdjustToMedia" order received                                     |
| EHD_ADJUSTING_STEP_2      | Sets height adjustment system position.                         | Width adjustment system is positioned                              |
| EHD_ADJUSTING_STEP_3      | No action executed                                              | Width adjustment system is positioned                              |

# EHD functionality description

[Specifications](https://confluence.efi.com/pages/viewpage.action?spaceKey=NSI&title=Edge+Hold+Down+in+14000Led)
```

### Program Logical/ExtPack/_Transport/EdgeHoldDown/EdgeHoldDownSim/EdgeHoldDownSim_v1/EdgeHoldDownSim (IEC)

#### EdgeHoldDownSim.st - Init, cyclic, exit code
```iecst
PROGRAM _INIT
	(* Insert code here *)

END_PROGRAM

PROGRAM _CYCLIC
	(* Insert code here *)
	data ACCESS ADR(gEdgeHoldDown);

END_PROGRAM

PROGRAM _EXIT
	(* Insert code here *)

END_PROGRAM
```

#### EdgeHoldDownSim.var - Local variables
```iecst
VAR
	data : REFERENCE TO EdgeHoldDown_typ;
END_VAR
```

### Program Logical/ExtPack/_Transport/JamDetectCtrl/JamDetect_v1/JamDetect (IEC)

#### JamDetectCtrl.var
```iecst
VAR
	JamDetect : REFERENCE TO JamDetect_typ;
	AlarmsReseted : JamDetectAlarms_typ;
	CommandsReseted : JamDetectCommands_typ;
	tonTestTimeOut : TON; (*Time to consider the test is wrong without an OK signal of the test*)
	tonTestsWaitAnswer : TON; (*Time to Start checking the result of the test*)
	tonNextTest : TON; (*Time to Wait for testing next device*)
	usiTestNum : USINT; (*Test number active*)
	iIndexSensor : USINT;
	ars_AlrJamDetectionSound : AutoResetSound;
	StatusPrevious : JamVibrationStatus_enum;
	xStatusChanged : BOOL;
	xTestFinished : BOOL;
	TestingStatus : JamTestingStatus_enum;
	xAnyCrashAlarm : BOOL;
	xAnyTestAlarm : BOOL;
END_VAR
VAR CONSTANT
	iHistoryLines : USINT := 20;
END_VAR
VAR
	StateHistory : ARRAY[0..iHistoryLines] OF JamVibrationStatus_enum;
	iIndexHistory : USINT;
END_VAR
VAR CONSTANT
	iTestingHistoryLines : USINT := 20;
END_VAR
VAR
	TestingStateHistory : ARRAY[0..iHistoryLines] OF JamTestingStatus_enum;
	iTestingIndexHistory : USINT;
	ctuConsecutiveLowJamDetected : ARRAY[0..1] OF CTU; (*Counter to check consecutive low jam detections*)
	tofConsecutiveLowJamDetected : ARRAY[0..1] OF TOF; (*Time to check consecutive low jam detections*)
	stWarningAlarmsLog : EventLog_typ;
	strAuxEventDesc : STRING[129];
END_VAR
```

#### EventLog.st
```iecst
ACTION LogWarningAlarm:

	stWarningAlarmsLog.Source := ELOG_TYPE_EHD;
	stWarningAlarmsLog.Severity:= ELOG_SEVERITY_INFO;
	stWarningAlarmsLog.Facility:= 0;
	stWarningAlarmsLog.ErrorCode:=0;

	IF ctuConsecutiveLowJamDetected[0].Q 	THEN 	stWarningAlarmsLog.Text := 'LowJamDetection > 3 in 1 min JDevice: ';
	ELSIF ctuConsecutiveLowJamDetected[1].Q THEN	stWarningAlarmsLog.Text := 'LowJamDetection > 10 in 30 min JDevice: ';
	END_IF

	brsftoa(iIndexJam, ADR(strAuxEventDesc));
	brsstrcat(ADR(stWarningAlarmsLog.Text), ADR(strAuxEventDesc));

	gEventLogLoader(EventData := ADR(stWarningAlarmsLog));

END_ACTION
```

#### JamTesting.st
```iecst
ACTION JamTesting:

	IF xStatusChanged THEN
		TestingStatus := JAMVIBT_INIT;
	END_IF

	(**TESTS ALARMS**)
	//All jam devices share the DO from PLC to test the sensors, 1 PLC DigitalOutput will activate the test of 1 sensor in all jam devices. So, never perform 2 tests simultaneously

	//Time to consider the test is wrong without an OK signal of the test
	tonTestTimeOut.IN := TestingStatus=JAMVIBT_CHECKING;
	tonTestTimeOut.PT := t#2s;
	tonTestTimeOut();

	//Time to Start checking the result of the test
	tonTestsWaitAnswer.IN := TestingStatus=JAMVIBT_WAITING_TO_CHECK;
	tonTestsWaitAnswer.PT := t#5s;
	tonTestsWaitAnswer();

	tonNextTest.IN := TestingStatus=JAMVIBT_GO_NEXT;
	tonNextTest.PT := t#300ms;
	tonNextTest();

	CASE TestingStatus OF

		JAMVIBT_INIT:
			usiTestNum := 1;
			TestingStatus := JAMVIBT_ACTIVATE_SIGNAL;

		JAMVIBT_ACTIVATE_SIGNAL:
			xTestFinished := FALSE;
			JamDetect.Outputs.xJamTestSignal[usiTestNum]:= JamDetect.Parameters.xBarInstalled[usiTestNum];
			TestingStatus := JAMVIBT_WAITING_TO_CHECK;

		JAMVIBT_WAITING_TO_CHECK:
			IF tonTestsWaitAnswer.Q THEN
				TestingStatus := JAMVIBT_CHECKING;
			END_IF

		JAMVIBT_CHECKING:
			IF NOT JamDetect.Inputs.xJamTestOk AND JamDetect.Parameters.xBarInstalled[usiTestNum] THEN
				JamDetect.Alarms.xAlrJamTest[usiTestNum] := TRUE;
			END_IF
			IF tonTestTimeOut.Q THEN
				JamDetect.Outputs.xJamTestSignal[usiTestNum]:= FALSE;
				TestingStatus := JAMVIBT_GO_NEXT;
			END_IF

		JAMVIBT_GO_NEXT:
			IF usiTestNum < JamDetect.Parameters.iSensorsQuantity THEN
				IF tonNextTest.Q THEN
					usiTestNum := usiTestNum + 1;
					TestingStatus := JAMVIBT_ACTIVATE_SIGNAL;
				END_IF
			ELSE
				xTestFinished := TRUE;
				TestingStatus := JAMVIBT_INIT;
			END_IF

	END_CASE

	//Saving state history
	IF TestingStatus<>TestingStateHistory[0] THEN
		FOR iTestingIndexHistory:=iTestingHistoryLines TO 1 BY -1 DO
			TestingStateHistory[iTestingIndexHistory]:=TestingStateHistory[iTestingIndexHistory-1];
		END_FOR
		TestingStateHistory[0]:=TestingStatus;
	END_IF

END_ACTION

ACTION ResetTestingOrders:

	xTestFinished := FALSE;

	FOR iIndexSensor:=1 TO JamDetect.Parameters.iSensorsQuantity BY 1 DO
		JamDetect.Outputs.xJamTestSignal[iIndexSensor]	:= FALSE;
	END_FOR

END_ACTION
```

### Program Logical/ExtPack/_Transport/JamDetectCtrl/JamDetect_v1/InitJamDetect (IEC)

#### InitJamDetect.st
```iecst
PROGRAM _CYCLIC
	iIndexJam:=1;
END_PROGRAM
```

- JamDocumentation.graphml - Block States graph (not shown)

### Program Logical/ExtPack/_Transport/JamDetectCtrl/JamDetectSim/JamDetectSim_v1/InitJamDetectSim

#### Cyclic.st
```iecst
PROGRAM _CYCLIC
	(* Insert code here *)
	usiJamDetectSimIndex := 1;

END_PROGRAM
```

### Program Logical/ExtPack/_Transport/NonCrashCtrl/NonCrashCtrl_v1/NonCrashCtrl

#### EventLog.st
```iecst
ACTION LogStopAlarm:

//	iReasonStop.0 := dataNC.Alarms.xAlrComsDrive;
//	iReasonStop.1 := dataNC.Alarms.xAlrDriveError;
//	iReasonStop.2 := dataNC.Alarms.xAlrOvertorque;
//	iReasonStop.3 := dataNC.Alarms.xAlrDiffContact;
//	iReasonStop.4 := dataNC.Alarms.xControllerNotReady;
//	iReasonStop.5 := dataNC.Alarms.xPerimeterNotDefined;
//	iReasonStop.6 := dataNC.Alarms.xGearBoxNotDefined;

	stEventLog.Source := ELOG_TYPE_NONCRASH;
	stEventLog.Severity:= ELOG_SEVERITY_INFO;
	stEventLog.Facility:= iIndexNonCrash;
	stEventLog.ErrorCode:=0;

	stEventLog.Text := 'Vacuum.LogStopAlarm';

	IF 		iReasonStop.0 THEN stEventLog.Text := 'Vacuum. xAlrComsMotor';
	ELSIF 	iReasonStop.1 THEN stEventLog.Text := 'Vacuum. xAlrDriveError';
	ELSIF 	iReasonStop.2 THEN stEventLog.Text := 'Vacuum. xAlrOvertorque';
	ELSIF 	iReasonStop.3 THEN stEventLog.Text := 'Vacuum. xAlrDiffContact';
	ELSIF 	iReasonStop.4 THEN stEventLog.Text := 'Vacuum. xControllerNotReady';
	ELSIF 	iReasonStop.5 THEN stEventLog.Text := 'Vacuum. xPerimeterNotDefined';
	ELSIF 	iReasonStop.6 THEN stEventLog.Text := 'Vacuum. xGearBoxNotDefined';
	END_IF

	gEventLogLoader(EventData := ADR(stEventLog));

END_ACTION
```

#### NonCrashCtrl.st
```iecst
PROGRAM _CYCLIC

	//References of the program
	dataNC ACCESS ADR (gNonCrash[iIndexNonCrash]);

	dataNC.Status.xInstalled := dataNC.Parameters.xInstalled;

	//Just defined as not installed when the NonCrash is stopped
	IF dataNC.Status.xInstalled THEN
		//Managing when not enabled the start or the error status. Not exiting while moving
		IF dataNC.parSw.xEnable THEN
			dataNC.Status.xEnabled := TRUE;
		ELSIF NOT dataNC.parSw.xEnable AND (StatusCtrl=NONCRASH_NOT_INITIALIZED OR StatusCtrl=NONCRASH_ERROR) THEN
			dataNC.Status.xEnabled := FALSE;
		END_IF
	END_IF

	IF NOT dataNC.Status.xInstalled OR NOT dataNC.Status.xEnabled THEN
		ResetAlarms;
		iIndexNonCrash:= iIndexNonCrash +1;
		RETURN;
	END_IF

	//Reference to the motor of the blower
	AxisMotor ACCESS ADR(gAxis[dataNC.Parameters.iIndexMotor]);

	//Limits of the movement data

	// Initial values in S1400
	//gNonCrash[1].Parameters.DriveUnit.LinealPerimeter.GearBox:=30;
	//gNonCrash[1].Parameters.DriveUnit.LinealPerimeter.Perimeter:=500;

	dataNC.Parameters.DriveUnit.LinealPerimeter.GearBox := MAX(dataNC.parSw.rGearBox, 0.001);
	dataNC.Parameters.DriveUnit.LinealPerimeter.Perimeter := MAX(dataNC.parSw.rPerimeter, 100);

	dataNC.parSw.rSpeedOffset := LIMIT(-1.0, dataNC.parSw.rSpeedOffset, 1.0);

	StateManager;

	Alarms;

	xRunningState := StatusCtrl=NONCRASH_RUNNING OR StatusCtrl=NONCRASH_RUN_ORDER;

	IF dataNC.Parameters.MotorDirection = MOTOR_NEGATIVE THEN
		AxisMotor.Parameter.Direction := MOTOR_NEGATIVE_AXIS;
	ELSE
		AxisMotor.Parameter.Direction := MOTOR_POSITIVE_AXIS;
	END_IF

	//Drive unit Managment
	DriveUnitManager.TransmissionData := dataNC.Parameters.DriveUnit;

	// Define the Status of the Motor with the Status of the Axis
	DriveUnitManager.PulsesSpeedDevice := AxisMotor.Status.ActVelocity;
	DriveUnitManager.Calculation := CALC_SPEED_MMIN;
	DriveUnitManager();
	dataNC.Status.Motor.rCurrentSpeed	:= ABS(DriveUnitManager.SpeedMminDevice);
	dataNC.Status.Motor.rCurrentSpeedUnits := ABS(AxisMotor.Status.ActVelocity);

	DriveUnitManager.AccelerationDesired := dataNC.Parameters.rAcceleration;
	DriveUnitManager.Calculation := CALC_ACC_PULSES;
	DriveUnitManager();
	AxisMotor.Parameter.Acceleration := MIN(DriveUnitManager.pulsesAccelerationDesired, AxisMotor.Status.MaxAccelerationNeg, AxisMotor.Status.MaxAccelerationPos);

	DriveUnitManager.DecelerationDesired := dataNC.Parameters.rDeceleration;
	DriveUnitManager.Calculation := CALC_DEC_PULSES;
	DriveUnitManager();
	AxisMotor.Parameter.Deceleration := MIN(DriveUnitManager.pulsesDecelerationDesired, AxisMotor.Status.MaxDecelerationNeg, AxisMotor.Status.MaxDecelerationPos);

	// Set velocity. Calculate speed in pulses with DriveUnit
	DriveUnitManager.SpeedMminDesired := MAX(dataNC.Parameters.rSpeedSetPoint + dataNC.parSw.rSpeedOffset,0.5); 	//It avoids a 0 speed and do not see a Continuous Movement state
	DriveUnitManager.Calculation := CALC_SPEED_MMIN_PULSES;
	DriveUnitManager();

	// Sending axis motion orders
	AxisMotor.Command.Move.Halt     := AxisMotor.Status.PLCopenState.ContinuousMotion AND NOT xRunningState;
	AxisMotor.Command.Move.Velocity := EDGEPOS(xRunningState) OR AxisMotor.Parameter.Speed <> DriveUnitManager.pulsesSpeedDesired; // JMH: It is important the order of these two lines
	AxisMotor.Parameter.Speed       := DriveUnitManager.pulsesSpeedDesired; // JMH: It is important the order of these two lines

	//Define the outputs of the Structure
	dataNC.Status.State := StatusCtrl;

	dataNC.Status.Motor.xRunning := AxisMotor.Status.PLCopenState.ContinuousMotion;
	dataNC.Status.Motor.rTorque := AxisMotor.Status.ActTorque;
	dataNC.Status.Motor.ErrorId := AxisMotor.Status.ErrorID;

	iIndexNonCrash := iIndexNonCrash + 1;

END_PROGRAM
```

### Program Logical/ExtPack/_Transport/NonCrashCtrl/NonCrashSim/NonCrashSim_v1/NonCrashSim (IEC)

#### Main.st - Init, cyclic, exit code
```iecst
PROGRAM _INIT

END_PROGRAM

PROGRAM _CYCLIC

	nonCrash ACCESS ADR(gNonCrash[iNonCrashSimIndex]);
	nonCrashSim ACCESS ADR(gSimNonCrash[iNonCrashSimIndex]);

	IF nonCrashSim.Commands.xRaiseAlrComsDrive THEN
		nonCrash.Alarms.xAlrComsDrive := TRUE;
	END_IF

	IF nonCrashSim.Commands.xRaiseAlrDiffContact THEN
		nonCrash.Alarms.xAlrDiffContact := TRUE;
	END_IF

	IF nonCrashSim.Commands.xRaiseAlrDriveError THEN
		nonCrash.Alarms.xAlrDriveError := TRUE;
	END_IF

	IF nonCrashSim.Commands.xRaiseAlrOvertorque THEN
		nonCrash.Alarms.xAlrOvertorque := TRUE;
	END_IF

	IF nonCrashSim.Commands.xRaiseControllerNotReady THEN
		nonCrash.Alarms.xControllerNotReady := TRUE;
	END_IF

	//Increase the index for simulating the next item
	iNonCrashSimIndex := iNonCrashSimIndex +1;

END_PROGRAM
```

#### NonCrashSim.var - Local variables
```iecst
VAR
	nonCrash : REFERENCE TO NonCrash_typ;
	nonCrashSim : REFERENCE TO SimNonCrash_typ;
END_VAR
```

### PairedIclaMotors.var
```iecst
VAR
	iIndexPairedIclaMotors : USINT;
END_VAR
```

- PairedIclaMotors.graphml (not shown)

### Program Logical/ExtPack/_Transport/PairedIclaMotors/PairedIclaMotors_v1/InitPairedIclaMotors

#### InitPairedIclaMotors.st
```iecst
PROGRAM _CYCLIC
	iIndexPairedIclaMotors := 1;
END_PROGRAM
```

### Program Logical/ExtPack/_Transport/PairedIclaMotors/PairedIclaMotors_v1/PairedIclaMotors
